# B&R Automation Studio project TD52 (part 44)

### Program Logical/Customized/c_red (IEC, version 4.11.0) - customisation task for exernal power reductions

#### c_redCyclic.st
```iecst
(*******************************************************************************
c_red 			customized power reductions

This code is confidential and proprietary to the INNIO Company.
It may not be used in any form, or reproduced in any manner,
without written permission of the INNIO Company.
Copyright, INNIO Company, 2021

Customized modifications: -
------------------------

History:
-------
V3.90.0	03.07.2012 Zengerer		new, (function moved from task gasum )
V4.02.0 ??.??.2015  ??			cleanup, separated INI file
V4.03.0	10.11.2015 Zengerer		cleanup
V4.04.0	08.03.2017 Zengerer		replace IN_CU.tCustAnaIn[1].Ai by a neutral IN_CU.tCustAnaIn[0].Ai default, to avoid conflicts when task is not used
V4.11.0	16.08.2021 Weitzer 		Delete W_XXmA constant variables

Instructions for use:
--------------------
connect var for customized spare power redutions

! ALL REDUCTIONS HAVE TO BE NORMED FROM 0 to 1 EQUALS 0 to P nominal

Outstandings:
------------
adopt this task according customer needs
replace [0] with actual used channel numbers IN_CU.tCustAnaIn[0].Ai;

*******************************************************************************)

PROGRAM _CYCLIC

	(*-----------------------------------------------------------------------------------------*)
	(*                                        TASK INPUTS                                      *)
	(*-----------------------------------------------------------------------------------------*)
 	OUT_CU.bP_Red_Sp_Lim1Act :=	FALSE;						(* CONNNECT REDUCTION ACTIVATION BIT HERE *)
	xSigScalR_Lim1Act.X := 		IN_CU.tCustAnaIn[0].Ai;		(* CONNNECT REDUCTION VALUE for customer spare power reduction, e.g. IN_CU.tCustAnaIn[1].Ai;	 *)
															(*hint: connect xSigScalR_Lim1Act.X1 and x2 also to available spare parameter*)

	OUT_CU.bP_Red_Sp_Lim2Act  	:= FALSE;					(* CONNNECT REDUCTION ACTIVATION BIT HERE *)
	xSigScalR_Lim2Act.X := 		IN_CU.tCustAnaIn[0].Ai;		(* CONNNECT REDUCTION VALUE for customer spare power reduction, e.g. IN_CU.tCustAnaIn[2].Ai; *)
															(*hint: connect xSigScalR_Lim2Act.X1 and x2 also to available spare parameter*)

	OUT_CU.bP_Red_Sp_Lim3Act  	:= FALSE;					(* CONNNECT REDUCTION ACTIVATION BIT HERE *)
	xSigScalR_Lim3Act.X := 		IN_CU.tCustAnaIn[0].Ai;		(* CONNNECT REDUCTION VALUE for customer spare power reduction, e.g. IN_CU.tCustAnaIn[3].Ai; *)
															(*hint: connect xSigScalR_Lim3Act.X1 and x2 also to available spare parameter*)

	(*-----------------------------------------------------------------------------------------*)
	(* Customer spare power reductions
	(*-----------------------------------------------------------------------------------------*)
	(* Reserve reduction #1 *)
	OUT_CU.bP_Red_Sp_Lim1Act; //:= FALSE;
	xSigScalR_Lim1Act.X; //		:= IN_CU.tCustAnaIn[x].Ai;
	xSigScalR_Lim1Act.X1 		:= Para.rCust_SparePara[0];		(* CONNNECT REDUCTION START VALUE, e.g. Para.rCust_SparePara[1]; *)
	xSigScalR_Lim1Act.Y1		:= 1.00;
	xSigScalR_Lim1Act.X2		:= Para.rCust_SparePara[0];		(* CONNNECT REDUCTION END VALUE, e.g. Para.rCust_SparePara[2];	 *)
	xSigScalR_Lim1Act.Y2		:= 0.50;
	xSigScalR_Lim1Act();
	IF OUT_CU.bP_Red_Sp_Lim1Act THEN
		OUT_CU.rP_Red_Sp_Lim1_Norm	:= LIMIT(0,xSigScalR_Lim1Act.Y_SCAL,1.0);
	ELSE
		OUT_CU.rP_Red_Sp_Lim1_Norm	:= 1.0;
	END_IF;

	(* Reserve reduction #2 *)
	OUT_CU.bP_Red_Sp_Lim2Act; //:= FALSE;
	xSigScalR_Lim2Act.X; //		:= IN_CU.tCustAnaIn[x].Ai;
	xSigScalR_Lim2Act.X1 		:= Para.rCust_SparePara[0];		(* CONNNECT REDUCTION START VALUE, e.g. Para.rCust_SparePara[1]; *)
	xSigScalR_Lim2Act.Y1		:= 1.00;
	xSigScalR_Lim2Act.X2		:= Para.rCust_SparePara[0];		(* CONNNECT REDUCTION END VALUE, e.g. Para.rCust_SparePara[2];	 *)
	xSigScalR_Lim2Act.Y2		:= 0.50;
	xSigScalR_Lim2Act();
	IF OUT_CU.bP_Red_Sp_Lim2Act THEN
		OUT_CU.rP_Red_Sp_Lim2_Norm	:= LIMIT(0,xSigScalR_Lim2Act.Y_SCAL,1.0);
	ELSE
		OUT_CU.rP_Red_Sp_Lim2_Norm	:= 1.0;
	END_IF;

	(* Reserve reduction #3 *)
	OUT_CU.bP_Red_Sp_Lim3Act; //:= FALSE;
	xSigScalR_Lim3Act.X	; //	:= IN_CU.tCustAnaIn[x].Ai;
	xSigScalR_Lim3Act.X1 		:= Para.rCust_SparePara[0];		(* CONNNECT REDUCTION START VALUE, e.g. Para.rCust_SparePara[1]; *)
	xSigScalR_Lim3Act.Y1		:= 1.00;
	xSigScalR_Lim3Act.X2		:= Para.rCust_SparePara[0];		(* CONNNECT REDUCTION END VALUE, e.g. Para.rCust_SparePara[2];	 *)
	xSigScalR_Lim3Act.Y2		:= 0.50;
	xSigScalR_Lim3Act();
	IF OUT_CU.bP_Red_Sp_Lim3Act THEN
		OUT_CU.rP_Red_Sp_Lim3_Norm	:= LIMIT(0,xSigScalR_Lim3Act.Y_SCAL,1.0);
	ELSE
		OUT_CU.rP_Red_Sp_Lim3_Norm	:= 1.0;
	END_IF;

	(*----------------------------------------------------------------------------------*)
	(* external utility(evu) request power reduction = iIdx_Pred_Type	:= neu25(31) *)
	(*----------------------------------------------------------------------------------*)
	(* Functionality MOVED TO MM GRID Code! *)

	(*----------------------------------------------------------------------------------*)
	(* limits for feedback signals to utility *)
	(*----------------------------------------------------------------------------------*)
	ton_RM_EVU[0](IN:= NOT IN_CU.tDI_Dem_P_Red_EVU_Stage1.Di AND NOT IN_CU.tDI_Dem_P_Red_EVU_Stage2.Di AND NOT IN_CU.tDI_Dem_P_Red_EVU_Stage3.Di AND IN_CU.bMCB_On , PT:= T#10s);	(* MCB_ON? -> to clarify...*)
	OUT_CU.tDO_P_Red_EVU_Stage0.Do := ton_RM_EVU[0].Q;		(* no power limit.and no lockout module *)

	lim_lo[1]( In:= IN_CU.rP_Act[1], Gw:= (Para.rP_Red_EVU_Stage1 + 0.01), Hy:= 0.01 );	(*OLD: lim_lo[1](In:= DINT_TO_INT((INT_TO_DINT(P_IST) * 1000)/ PN_GASART), Gw:= (ssPowRed_Utility_1 +10), Hy:= 10);*)
	ton_RM_EVU[1]( IN:= lim_lo[1].Q AND IN_CU.tDI_Dem_P_Red_EVU_Stage1.Di, PT:= T#30s );	(**)
	OUT_CU.tDO_P_Red_EVU_Stage1.Do := ton_RM_EVU[1].Q;		(* power limit.stage 1 (small reduction) *)

	lim_lo[2]( In:= IN_CU.rP_Act[1], Gw:= (Para.rP_Red_EVU_Stage2 + 0.01), Hy:= 0.01 );  (*OLD: lim_lo[2](In:= DINT_TO_INT((INT_TO_DINT(P_IST) * 1000)/ PN_GASART), Gw:= (ssPowRed_Utility_2 +10), Hy:= 10);*)
	ton_RM_EVU[2]( IN:= lim_lo[2].Q AND IN_CU.tDI_Dem_P_Red_EVU_Stage2.Di, PT:= T#30s );	(**)
	OUT_CU.tDO_P_Red_EVU_Stage2.Do := ton_RM_EVU[2].Q;		(* power limit.stage 2 (more reduction) *)

	lim_lo[3]( In:= IN_CU.rP_Act[1], Gw:= (Para.rP_Red_EVU_Stage3 + 0.01), Hy:= 0.01 );  (*OLD: lim_lo[3](In:= DINT_TO_INT((INT_TO_DINT(P_IST) * 1000)/ PN_GASART), Gw:= (ssPowRed_Utility_3 +10), Hy:= 10);*)
	ton_RM_EVU[3]( IN:= lim_lo[3].Q AND IN_CU.tDI_Dem_P_Red_EVU_Stage3.Di, PT:= T#30s );	(**)
	OUT_CU.tDO_P_Red_EVU_Stage3.Do := ton_RM_EVU[3].Q;		(* power limit.stage 3 (more reduction) *)

	lim_lo[4]( In:= IN_CU.rP_Act[1], Gw:= (Para.rP_Red_EVU_Stage4 + 0.01), Hy:= 0.01 );  (*OLD: lim_lo[4](In:= DINT_TO_INT((INT_TO_DINT(P_IST) * 1000)/ PN_GASART), Gw:= (ssPowRed_Utility_4 +10), Hy:= 10);*)
	ton_RM_EVU[4]( IN:= lim_lo[4].Q AND IN_CU.tDI_Dem_P_Red_EVU_Stage4.Di, PT:= T#30s );	(**)
	OUT_CU.tDO_P_Red_EVU_Stage4.Do := ton_RM_EVU[4].Q;		(* power limit.stage 4 (more reduction) *)

	lim_lo[5]( In:= IN_CU.rP_Act[1], Gw:= (Para.rP_Red_EVU_Stage5 + 0.01), Hy:= 0.01 );  (*OLD: lim_lo[?6?](In:= DINT_TO_INT((INT_TO_DINT(P_IST) * 1000)/ PN_GASART), Gw:= (ssPowRed_Utility_5 +10), Hy:= 10);*)
	ton_RM_EVU[5]( IN:= lim_lo[5].Q AND IN_CU.tDI_Dem_P_Red_EVU_Stage5.Di, PT:= T#30s );	(**)
	OUT_CU.tDO_P_Red_EVU_Stage5.Do := ton_RM_EVU[5].Q;		(*  (=most reduction)*)

	(*------------------------------------------------------------------------------------------*)
	(* generator: power factor controller dependent power reductions ??							*)
	(*------------------------------------------------------------------------------------------*)
	(* FUNCTION MOVED TO MODUL GENERATOR! *)

	(*-----------------------------------------------------------------------------------------*)
	(* power reduction for Extern – Analog (analog_dp):
	(*-----------------------------------------------------------------------------------------*)

	IF IN_CU.rP_Nom > 0 THEN
		rP_Red_AI_Norm := IN_CU.tP_Red_AI_Norm.Ai / IN_CU.rP_Nom;		(* parameter are entered in KW, so convert setpoint to Norm here    *)
	ELSE
		rP_Red_AI_Norm := 1.0;
	END_IF
			(* scaling (DISABELED HERE! NO additional scaling, allready done in the HAL (with customized parameter) *)
			Para.rI_P_Red_AI_NormScalMin;	Para.rI_P_Red_AI_NormScalMax;
			Para.rP_Red_AI_NormScalMin;		Para.rP_Red_AI_NormScalMax;

	(* power reduction on RSS Remote: (AFW_F)*)
	IF (IN_CU.iIdx_RSS = 2) AND IN_CU.tP_Red_AI_Norm.GoodQual THEN		(* locale representation of old AWS_F from IN_CU.iIdx_RSS = 2  *)
		OUT_CU.rP_Red_AI_Norm := LIMIT(0.5, rP_Red_AI_Norm, 1.0);		(*= analog power limit value *)
		OUT_CU.bP_Red_AI_Enable := TRUE ;
	ELSE
		OUT_CU.rP_Red_AI_Norm := 1.0;
		OUT_CU.bP_Red_AI_Enable := FALSE ;
	END_IF

	(*-----------------------------------------------------------------------------------------*)
	(*                                        TASK OUTPUTS                                     *)
	(*-----------------------------------------------------------------------------------------*)
	(* Prototype usage of all outputs: *)
	OUT_CU.bP_Red_Sp_Lim1Act ; 		(* power setpoint limit 1 activ *) (*OldName: bPowerSetpointLimit1; Cycle: 5;*)
	OUT_CU.bP_Red_Sp_Lim2Act ; 		(* power setpoint limit 2 activ *) (*OldName: bPowerSetpointLimit2; Cycle: 5;*)
	OUT_CU.bP_Red_Sp_Lim3Act ; 		(* power setpoint limit 3 activ *) (*OldName: bPowerSetpointLimit3; Cycle: 5;*)
	OUT_CU.rP_Red_Sp_Lim1_Norm ; 	(* power setpoint limit 1  related to rP_Nom *) (*OldName: ssPowerSetpointLimit1; Cycle: 5;*)
	OUT_CU.rP_Red_Sp_Lim2_Norm ; 	(* power setpoint limit 2  related to rP_Nom] *) (*OldName: ssPowerSetpointLimit2; Cycle: 5;*)
	OUT_CU.rP_Red_Sp_Lim3_Norm ; 	(* power setpoint limit 3  related to rP_Nom *) (*OldName: ssPowerSetpointLimit3; Cycle: 5;*)
	OUT_CU.bP_Red_EVU_Enable ; 		(* *) (*OldName: RED_EVU_Aktiv; Cycle: 5;*)
	OUT_CU.rP_Red_EVU_Norm ; 		(* power redutcion by utility *) (*OldName: RED_EVU; Cycle: 5;*)
	OUT_CU.rP_Red_AI_Norm ; 		(* power reduction by analog input *) (*OldName: ssPowerRedAnalog; Cycle: 5;*)

END_PROGRAM
```

#### c_redInit.st
```iecst
(********************************************************************
 * COPYRIGHT -- INNIO Company
 ********************************************************************
 * Programm: c_red
 * Datei: c_redInit.st
 * Autor: ZengereS
 * Erstellt: 24.Juni 2015
 ********************************************************************)

PROGRAM _INIT

	OUT_CU.rP_Red_EVU_Norm := 	1.0;	(*	ssExtPwrSetP4 ? *)

	OUT_CU.rP_Red_AI_Norm := 	1.0; 	(* power reduction by analog input *) (*OldName: ssPowerRedAnalog *)

	(* This factory default definition is only a backuü fallback solution. *)
	(* Set parameter values for normal operation in parameter file! *)
	ParaFactoryDefault.rP_Red_EVU_Stage1 := 		0.1;	(* [1/ P nom] *)
	ParaFactoryDefault.rP_Red_EVU_Stage2 := 		0.2;	(* [1/ P nom] *)
	ParaFactoryDefault.rP_Red_EVU_Stage3 := 		0.3;	(* [1/ P nom] *)
	ParaFactoryDefault.rP_Red_EVU_Stage4 := 		0.4;	(* [1/ P nom] *)
	ParaFactoryDefault.rP_Red_EVU_Stage5 := 		0.5;	(* [1/ P nom] *)

END_PROGRAM
```

#### c_red.var - Lokale Variablen
```iecst
(********************************************************************
 * COPYRIGHT -- INNIO Company
 ********************************************************************
 * Programm: c_red
 * Datei: c_red.var
 * Autor: ZengereS
 * Erstellt: 20. Februar 2013
 ********************************************************************
 * Lokale Variablen des Programms c_red
 ********************************************************************)
VAR
	ton_RM_EVU : ARRAY[0..5] OF TON;
	lim_lo : ARRAY[0..5] OF GR_MAXR;
	rP_Red_AI_Norm : REAL;
	xSigScalR_Lim1Act : xSigScal_R;
	xSigScalR_Lim2Act : xSigScal_R;
	xSigScalR_Lim3Act : xSigScal_R;
END_VAR
```

### Program Logical/Customized/c_set (IEC, version 4.13.0) - customisation task for external power setpoints

#### c_setCyclic.st
```iecst
(*******************************************************************************
c_set 			customized power SETPOINTS

This code is confidential and proprietary to the INNIO Company.
It may not be used in any form, or reproduced in any manner,
without written permission of the INNIO Company.
Copyright, INNIO Company, 2023

Customized modifications: -
------------------------

History:
-------
								History cleanup, Version based on V4.02.1	04.03.2015: prepared interface FOR different PI timing (->Caks Michael)
V4.03.0	12.11.2015 Zengerer		P_Set_ExtAI_Norm  changed fallback logic; REACTIVETED DI POWER SETPOINT LOGIC AND PARAMETER HERE! (since code IN GRID CODE task statGR HAS GOT A DIFFERENT FUNCTIONALITY
		22.12.2015 Ze/Caks		Para.bCA_IgnP_CylOffset_Active
V4.04.1 05.09.2017 zengerer		Nachziehen der Netzbezugsregler Änderungen von Schwab Christoph / Caks Michael aus File Bugs&Solution_MnsCtrl.zip
V4.04.5 10.10.2017 Zengerer		Update with interfaces from BASISUPDATE 4.04.00.05 iIdx_Pred_Type State
V4.05.0 10.10.2017 zengerer		prepared interface for adopted gasmixing setpoint at testbench or for customized applications
V4.05.1 07.03.2018 zengerer		cleanup
		30.01.2019 Hohensinner	added new interfaces to OP and GC
		20.03.2019 Hohensinner	Added external controller interface
V4.07.1	03.04.2019 Hohensinner	Added Parameter Info for new interfaces and comments
V4.09.0 22.01.2020 zengerer		avoid P setpoint switching with 0mA Value:	(IN_CU.tP_Set_ExtAI_Norm.GoodQual OR Para.rI_P_Set_ExtAI_NormScalMin < 0.004)
V4.10.0	16.10.2020 Weitzer 		Release of custom GCB synchronization demand OUT_CU.bCust_Dem_Sy and MCB re-synchronization demand OUT_CU.bCust_Dem_RSy added
		19.01.2021 Weitzer		Custom synchronization blocking added (OUT_CU.bBloc_SY_Rel_Cust)
		27.01.2021 Zengerer		TOF_N_Set_ExtAI_Norm_GoodQual T#12s delay,
		28.01.2021 Zengerer		power setpoint range limitation min #53
		12.03.2021 Zengerer		#262- Conditions internal or bus speed setpoint active for speed offset:	AND	(IN_CU.iMsg[2136]>0 OR IN_CU.iMsg[2137]>0)
V4.10.1	xx.08.2021 Ze, GruberK.	Issue #530 ...need N_Offset and not external setpoint; limit value to parameter values
V4.11.0	16.08.2021 Keller		External Droop Power setpoint (AI, Bus), iSource_F_N_OffsSet
V4.11.0	16.08.2021 Weitzer 		Delete W_XXmA constant variables
		21.01.2022 MayerR	    AI scaling and signal source selection for OUT_CU.rUset_Isl moved to GC module(v_ctr) and Bus interfaces (OUT_CU.rUset_Isl_Bus and OUT_CU.rQset_Droop_Bus) added
V4.11.1 31.05.2022 lettenb.		default setting OUT_CU.bCust_Dem_RSy := TRUE -> FALSE(RSy only in case of customer demand), bugfix
V4.12.0 22.01.2023 Zuschnig		H2 content via bus added
V4.13.0	25.05.2023 Zengerer 	Speed Setpoint limitation #1106
		24.08.2023 Zengerer		IN_CU.bMsg[xxxx] introduced
		16.10.2023 Bachler  	add OUT_CU.bOtherGeneratorsInLSL for bumpless transition to LSL
		20.11.2023 Farre		interfaces to SY, OP, GC, GR needed for Microgrid applications (2023-168)
		29.11.2023 Goenczi		add new interfaces to SY and OP

Instructions for use:
--------------------
connect var's for customized power setpoints

! ALL SETPOINTS HAVE TO BE NORMED FROM 0 to 1 EQUALS 0 to P nominal

Outstandings:
------------
TODO: CHECK NEW CUSTOMISED PARA vvm/addPLCtag

  adopt this task according customer needs

! Be aware, that several setpoints are also influenced from GRID CODE MODULE, if this is engaged !

*******************************************************************************)

PROGRAM _CYCLIC

	(*----------------------------------------------------------------------------------*)
	(* external DI request power setpoints *) (*REACTIVETED SETPOINT LOGIC AND PARAMETER HERE! (since code IN GRID CODE task statGR HAS GOT A NEW FUNCTIONALITY *)
	(*----------------------------------------------------------------------------------*)
	(* power setpoint according external request digital inputs *)
	IF    IN_CU.tP_GenC_SetFix5EU.Di	THEN
		OUT_CU.rP_Set_ExtDI_Cust_Norm	:=	LIMIT(0.4, Para.rP_Set5_ExtDI_Norm, 1.0); 	(*OldName: AW_EXPSH_DI; Cycle: 5;*)
	ELSIF IN_CU.tP_GenC_SetFix4EU.Di	THEN
		OUT_CU.rP_Set_ExtDI_Cust_Norm	:=	LIMIT(0.4, Para.rP_Set4_ExtDI_Norm, 1.0);
	ELSIF IN_CU.tP_GenC_SetFix3EU.Di	THEN
		OUT_CU.rP_Set_ExtDI_Cust_Norm	:=	LIMIT(0.4, Para.rP_Set3_ExtDI_Norm, 1.0);
	ELSIF IN_CU.tP_GenC_SetFix2EU.Di	THEN
		OUT_CU.rP_Set_ExtDI_Cust_Norm	:=	LIMIT(0.4, Para.rP_Set2_ExtDI_Norm, 1.0);
	ELSIF IN_CU.tP_GenC_SetFix1EU.Di	THEN
		OUT_CU.rP_Set_ExtDI_Cust_Norm	:=	LIMIT(0.4, Para.rP_Set1_ExtDI_Norm, 1.0);
	ELSE
		OUT_CU.rP_Set_ExtDI_Cust_Norm	:=	1.0;										(* replacement for rP_Set_ExtDI_Norm *)
	END_IF;

	OUT_CU.bP_Set_ExtDI_Enable := 	IN_CU.tP_GenC_SetFix1EU.Di OR
									IN_CU.tP_GenC_SetFix2EU.Di OR
									IN_CU.tP_GenC_SetFix3EU.Di OR
									IN_CU.tP_GenC_SetFix4EU.Di OR
									IN_CU.tP_GenC_SetFix5EU.Di;		(* or connect customized?*)

	(* power setpoint *)
	(******************)
	IF Para.bCtr_Mns_Enable AND IN_CU.tDem_Ctr_Mns.Di THEN
		rP_Set_ExtAI_Norm := OUT_CU.rP_Set_Mns_Norm;				(*old compatibility version, only for EngineController without rP_Set_Ctr_Mns_Norm*)
		OUT_CU.rP_Set_Ctr_Mns_Norm := OUT_CU.rP_Set_Mns_Norm;	(*new Interface V4.5, (in use for Ctr_Mns from V4.5 on)*)
		OUT_CU.bP_Set_Ctr_Mns_Enable := TRUE;					(*new Interface V4.5, (in use for Ctr_Mns from V4.5 on)*)
	ELSIF	IN_CU.rP_Nom > 0 THEN
		rP_Set_ExtAI_Norm := IN_CU.tP_Set_ExtAI_Norm.Ai / IN_CU.rP_Nom;		(* parameter are entered in KW, so convert Setpoint to Norm    *)
		OUT_CU.rP_Set_Ctr_Mns_Norm := rP_Set_ExtAI_Norm;
		OUT_CU.bP_Set_Ctr_Mns_Enable := FALSE;
	ELSE
		rP_Set_ExtAI_Norm := 1.0;
		OUT_CU.rP_Set_Ctr_Mns_Norm := rP_Set_ExtAI_Norm;
		OUT_CU.bP_Set_Ctr_Mns_Enable := FALSE;
	END_IF
			(* scaling (DISABELED HERE! NO additional scaling here, allready done in the HAL (with this customized parameter) *)
				Para.rI_P_Set_ExtAI_NormScalMin;	Para.rI_P_Set_ExtAI_NormScalMax;
				Para.rP_Set_ExtAI_NormScalMin;		Para.rP_Set_ExtAI_NormScalMax;

	IF 	(IN_CU.iIdx_OMSS = 2) AND 										(* =operating switch AUTO *)
		(IN_CU.iIdx_RSS = 2) AND 										(* =remote service selected *)
		(IN_CU.tP_Set_ExtAI_Norm.GoodQual								(* =analog input signal is ok *)
		  OR Para.rI_P_Set_ExtAI_NormScalMin < 0.004)
	THEN 																(* BWS_A AND Remote AND signal check is ok AND <deleted> *)
		OUT_CU.rP_Set_ExtAI_Norm := LIMIT(0.4,rP_Set_ExtAI_Norm, 1.0);	(*= analog power setpoint range limitation (V4.10 changed min)*)
		OUT_CU.bP_Set_ExtAI_Enable := TRUE ; 	 						(*OldName: AW_EXPSH_AI; Cycle: 5;*)
	ELSE
		OUT_CU.rP_Set_ExtAI_Norm := 0.50;								(*V4.03: changed fallback logic to standard min. load point*)
		OUT_CU.bP_Set_ExtAI_Enable := FALSE; 							(*OldName: AW_EXPSH_AI; Cycle: 5;*)
	END_IF

	(* speed setpoint *)
	(******************)
	IF Para.rN_EngNom > 0 THEN
		rN_Set_ExtAI_Norm := IN_CU.tN_Set_ExtAI_Norm.Ai / Para.rN_EngNom;		(* parameter are entered in KW, so convert Setpoint to Norm    *)
	ELSE
		rN_Set_ExtAI_Norm := 1.0;
	END_IF
			(* scaling (DISABELED HERE! No additional scaling here, allready done in the HAL (with this customized parameter) *)
			Para.rI_N_Set_ExtAI_NormScalMin;	Para.rI_N_Set_ExtAI_NormScalMax;
			Para.rN_Set_ExtAI_NormScalMin; 		Para.rN_Set_ExtAI_NormScalMax;

	TOF_N_Set_ExtAI_Norm_GoodQual(IN := IN_CU.tN_Set_ExtAI_Norm.GoodQual, PT := T#12s);		(*V4.10 delay*)
	IF  (IN_CU.iIdx_OMSS = 2) AND
		(IN_CU.iIdx_RSS = 2) AND
		TOF_N_Set_ExtAI_Norm_GoodQual.Q AND NOT
		(OUT_CU.iSource_F_N_OffsSet = 2) 			// typicaly needed N_Offset, not the external setpoint of previous default													(*V4.10 delay*)
//		IN_CU.tN_Set_ExtAI_Norm.GoodQual
// 		AND (Para.rI_N_Set_ExtAI_NormScalMin >0.004)
	THEN
		OUT_CU.rN_Set_ExtAI_Norm := LIMIT(0.9, rN_Set_ExtAI_Norm, 1.05);	(*= analog speed offset limitation  Limits adopted acc. issue #1106, 2023*)
		OUT_CU.bN_Set_ExtAI_Enable := TRUE ; (* *) 					(*OldName: AW_EX?SH_AI; Cycle: 5;*)
	ELSE
		OUT_CU.rN_Set_ExtAI_Norm := 1.0;
//		OUT_CU.bN_Set_ExtAI_Enable := FALSE ; (* *) 				(*OldName: AW_EX?SH_AI; Cycle: 5;*)
		OUT_CU.bN_Set_ExtAI_Enable := xOpMode.Island AND (Para.rI_N_Set_ExtAI_NormScalMin >0.004) AND TOF_N_Set_ExtAI_Norm_GoodQual.Q AND (OUT_CU.iSource_F_N_OffsSet = 2);  // Gruber K. - we need N_Offset and not external setpoint

	END_IF
				IN_CU.iMsg[2136]	;	(*display response: B2136 internal speed setpoint *)
 				IN_CU.iMsg[2137]	;	(*display response: B2137 external speed setpoint(bus) *)
				IN_CU.iMsg[2138]	;	(*display response: B2138 external speed setpoint(analoge) *)

	(******************************************************)
	(* Leistungsgrenzwert 1 - Customized z.b. ?Anforderung Lastabwurf? *)
	(*FEHLT NOCH:	GW_PGW1	   := DINT_TO_INT((INT_TO_DINT(PN_GASART) * Z_GW_PGW1  + 500) / 1000); *)
	Para.rP_Custom1_Norm_LimHi;		(* rP_Lim_Custom1_Norm == Z_GW_PGW1 = Para-Leistung-Grenzwerte-GRENZWERT 1 *)
	Para.rP_Custom1_Norm_HyHi;		(*FEHLT NOCH: 	HY_PGW1 ? Vorschlag  *)

(*FEHLT NOCH:	LAST_ABW :=  ( M_GSEIN AND NOT NS_EIN AND GW_PGW1 ) OR BL_OUT; *)	(*aus task pb8 -> wohin damit?*)

	(******************************************************)
	(* forwarding the parameter for different ignition timing on individual cylinders at testbench or for customized applications *)
	FOR ucCylinderCount := 1 TO 24 DO    (* bSetIndivTim can be used for tests                      *)
		IF IN_CU_ThisPlant.bCA_IgnP_ActiveMDE AND NOT IN_CU_ThisPlant.bMsg7000 THEN
			OUT_CU.rCA_IgnP_CylOffset[ucCylinderCount] := IN_CU_ThisPlant.rCA_IgnP_CylOffset_MDE[ucCylinderCount] * BOOL_TO_REAL(IN_CU_ThisPlant.bCA_IgnP_CylOffset_Active_MDE);
		ELSE
			OUT_CU.rCA_IgnP_CylOffset[ucCylinderCount] := Para.rCA_IgnP_CylOffset[ucCylinderCount] * BOOL_TO_REAL(Para.bCA_IgnP_CylOffset_Active);
		END_IF
	END_FOR

	(******************************************************)
	(* prepared interface for different PI timing on individual cylinders at testbench or for customized applications *)
     	OUT_CU.rCA_PI_Dur_COffset[1] := 0; 		(* custom PI duration offset cyl.1  *) (* OldName: ssTestBenchOffset *)
     	OUT_CU.rCA_PI_Dur_COffset[24] := 0; 	(* custom PI duration offset cyl.24 *) (* OldName: ssTestBenchOffset *)

	(******************************************************)
	(* prepared interface for adopted gasmixing setpoint *)
		OUT_CU.bOptGT_RatioMix_Set 	:= FALSE;   //:= TRUE;
 		OUT_CU.rGT_RatioMix_Set;				(* Fuel blending setpoint -> 0 - 1 = 0 - 100% )

	(******************************************************)

	(*** Enable bit for external speed / voltage controller ***)
	OUT_CU.bExtCtrOk := NOT IN_CU.tExtCtrOk.GoodQual OR IN_CU.tExtCtrOk.Di;		(* DI for use with ComAp or another external speed / voltage controller *)

	(*** Reactive power setpoint for voltage droop mode ***)
	(* Conversion:		1.0					100%Snom		*)
	(* Value range:		-1.0 to 1.0		-100% to 100%Snom	*)
	(* Build in Ramp:	0.01/s				1%Unom/s   		*)
	(* Enable:			Parameter 14298 must be set to 1	*)
	(* Droop gradient:	Parameter 14299						*)
	OUT_CU.rQset_Droop_Bus;									(* External reactive power setpoint for frequency droop mode over Bus - for project specific usage *)

	(* Voltage setpoint in Isolated operation, 0= no setpoint, 1= Droop, 2= External *)
	OUT_CU.rUset_Isl_Bus;									(* External Voltage setpoint (Island operation) over Bus - for project specific usage *)

	(*** Speed offset setpoint in Isolated operation ***)
	(* Conversion:		1.0					1 rpm			*)
	(* Value range:		-50	to +50			-50 to +50 rpm	*)
	(* Enable:			Parameter 14300 must be set to 2	*)
	IF IN_CU.tN_Set_ExtAI_Norm.GoodQual AND OUT_CU.bExtCtrOk THEN
		(* Check if value --> -50 to +50, Parameter 11781 should be -50 rpm & 11780 should be +50 rpm  *)
		IF		Para.rN_Set_ExtAI_NormScalMax < 150.0
			AND	Para.rN_Set_ExtAI_NormScalMin > -150.0
			//AND	(IN_CU.iMsg[2136]>0 OR IN_CU.iMsg[2137]>0)	// Gruber K. - will not work with this line included		(*V4.10: Offset allowed only at internal(2136) or bus(2137) speed setpoint, to avoid duplicate speed reduction in case of alternative input use *)
			AND NOT(IN_CU.tN_Set_ExtAI_Norm.Ai < -rN_Set_ExtAI_Limit OR IN_CU.tN_Set_ExtAI_Norm.Ai > rN_Set_ExtAI_Limit)(*V4.11: plausibility check *)
			THEN
				OUT_CU.rN_Offs_Cust		:=	LIMIT(Para.rN_Set_ExtAI_NormScalMin, IN_CU.tN_Set_ExtAI_Norm.Ai, Para.rN_Set_ExtAI_NormScalMax); (*Gruber K. - limit vlaue to parameter values*)
			(* Check if value --> 1450 to 1550, Parameter 11781 should be 0 or 1450 rpm & 11780 should be 1550 rpm *)
		ELSIF Para.rN_Set_ExtAI_NormScalMax > Para.rN_EngNom * 0.9 AND Para.rN_Set_ExtAI_NormScalMin < Para.rN_EngNom
			AND NOT(IN_CU.tN_Set_ExtAI_Norm.Ai < Para.rN_EngNom-rN_Set_ExtAI_Limit OR IN_CU.tN_Set_ExtAI_Norm.Ai > Para.rN_EngNom+rN_Set_ExtAI_Limit)(*V4.11: plausibility check *)
			THEN
			OUT_CU.rN_Offs_Cust		:=	IN_CU.tN_Set_ExtAI_Norm.Ai - Para.rN_EngNom;
			(* or implement your own solution *)							(* modify here if customer needs special scaling *)
		ELSE															(* modify here if customer needs special scaling *)
			OUT_CU.rN_Offs_Cust		:=	0.0;							(* modify here if customer needs special scaling *)
		END_IF
	ELSIF FALSE (*bN_OffsExt_Bus*) THEN									(* modify here if customer needs signal over bus *)
		OUT_CU.rN_Offs_Cust		:=	0.0;	(*rN_OffsExt_Bus*)			(* modify here if customer needs signal over bus *)
	ELSE
		OUT_CU.rN_Offs_Cust		:=	0.0;
	END_IF

	(*** Power setpoint for speed/frequency droop mode ***)
	(* Conversion:		1.0					100%Pnom		*)
	(* Value range:		0.0	to 1.0			0% to 100%Pnom	*)
	(* Build in Ramp:	Parameter 12095 & 13373	in %Pnom/s	*)
	(* Enable:			Parameter 14300 must be set to 1	*)
	(* Droop gradient:	Parameter 12109						*)
	OUT_CU.bP_Droop_Set_Bus;									(* Enable Droop power setpoint by Bus (if both true: has priority over AI)*)
	OUT_CU.bP_Droop_Set_AI; 									(* Enable Droop power setpoint by Analog input *)

	(** Fallback for power setpoint **)
	(* fallback if bP_Droop_Set_Bus = TRUE AND bus communication not OK *)
	(* fallback if bP_Droop_Set_AI = TRUE AND tP_Droop_Set.GoodQual = FALSE *)
	(* selection fallback mode, 0: default Para, 1: freeze last value*)
	OUT_CU.iIdx_Droop_SetDefaultCase 	:= Para.iIdx_Droop_SetDefaultCase;
	OUT_CU.rP_Set_Default_Norm 			:= Para.rP_Set_Default_Norm;

	(* Bus *)
	OUT_CU.rP_Droop_Set_Bus_Norm;(* HERE: implementation Droop setpoint bus interface *)
	IF NOT(IN_CU.bMsg[1147] OR IN_CU.bMsg[1099]) AND NOT(OUT_CU.rP_Droop_Set_Bus_Norm < -0.1 OR OUT_CU.rP_Droop_Set_Bus_Norm > 1.5) THEN
		rP_Droop_Set_Bus_old_Norm 		:= OUT_CU.rP_Droop_Set_Bus_Norm; 		(* save last valid setpoint *)
	ELSIF OUT_CU.iIdx_Droop_SetDefaultCase = 0 THEN
		OUT_CU.rP_Droop_Set_Bus_Norm	:= OUT_CU.rP_Set_Default_Norm;			(* 0: fallback, default parameter *)
	ELSIF OUT_CU.iIdx_Droop_SetDefaultCase = 1 THEN
		OUT_CU.rP_Droop_Set_Bus_Norm	:= rP_Droop_Set_Bus_old_Norm;			(* 1: fallback, freeze last valid setpoint *)
	ELSE
		OUT_CU.rP_Droop_Set_Bus_Norm	:= OUT_CU.rP_Set_Default_Norm;
	END_IF;

	(* Analog input *)
	IF IN_CU.tP_Droop_Set.GoodQual AND NOT(IN_CU.tP_Droop_Set.Ai < -0.1 OR IN_CU.tP_Droop_Set.Ai > 1.5) THEN
		OUT_CU.rP_Droop_Set_AI_Norm 	:= IN_CU.tP_Droop_Set.Ai;
		rP_Droop_Set_AI_old_Norm		:= OUT_CU.rP_Droop_Set_AI_Norm;  		(* save last valid setpoint *)
	ELSIF OUT_CU.iIdx_Droop_SetDefaultCase = 0 THEN
		OUT_CU.rP_Droop_Set_AI_Norm		:= OUT_CU.rP_Set_Default_Norm;			(* 0: fallback, default parameter *)
	ELSIF OUT_CU.iIdx_Droop_SetDefaultCase = 1 THEN
		OUT_CU.rP_Droop_Set_AI_Norm		:= rP_Droop_Set_AI_old_Norm;			(* 1: fallback, freeze last valid setpoint *)
	ELSE
		OUT_CU.rP_Droop_Set_AI_Norm 	:= OUT_CU.rP_Set_Default_Norm;
	END_IF;

	(* Load Sharing Mode, 0= no setpoint, 1= Droop, 2= External, 3= LSL *)
	OUT_CU.iSource_F_N_OffsSet := Para.iSource_F_N_OffsSet;
	MM2VIS.iSource_F_N_OffsSet := OUT_CU.iSource_F_N_OffsSet;

	(* Other Generators In Load Sharing Line *)
	(* If TRUE: 		Other engines are participating in the load sharing line *)
	(* Info: 			If this input is not provided a non smooth transition between LSL and the other load sharing modes will happen *)
	OUT_CU.bOtherGeneratorsInLSL;

	(*** Custom Engine demand ***)
	(* If TRUE:			Engine is demanded in AUTO & REMOTE	*)
	(* Info:			Add an Operating message why the engine is being demanded *)
	OUT_CU.bCust_Dem;

	(*** Custom Engine blocked ***)
	(* If TRUE:			Engine is blocked					*)
	(* Info:			If you want to block engine only in Stop mode use: 'bYourBit AND NOT bEng_StaSpdExc' *)
	OUT_CU.bEng_Block_Customized;

	(*Custom Emergency Power Supply release/demand*)

	(*** Release Island bit via Bus coupling ***)
	(* If FALSE:		Release island is blocked						*)
	(* Info:			Default value must be TRUE *)
	OUT_CU.bRel_I_Bus := TRUE;

	(*** Custom Release Island bit ***)
	(* If FALSE:		Release island is blocked						*)
	(* Info:			Default value must be TRUE *)
	OUT_CU.bCust_Rel_I := TRUE;

	(*** Custom Release Island operation busbar condition (if FALSE, mains cut-off with gcb) ***)
	(* If TRUE:			VKE10 condition TRUE					*)
	(* Info:			DO NOT CONFUSE WITH bRel_I Release island external bit!!! --- Default value must be FALSE *)
	OUT_CU.bCust_RelI_BB := FALSE;

	(*** Custom Emergency Power supply demand SY modul ***)
	(* If TRUE:			Additional demand condition to change to EPS mode in SY/sy_out task				*)
	(* Info:			Default value must be TRUE *)
	OUT_CU.bCust_Dem_EPS_Sy := TRUE;

	(*** External Emergency Power supply demand from Bus ***)
	(* If TRUE:			Emergency Power supply ON				*)
	(* Info:			Default value must be FALSE *)
	OUT_CU.bEng_Dem_EPS_Bus := FALSE;

	(*** Smooth engine discharge in multi engines island mode ***)
	(* If TRUE:			Engine is not demanded for island, request auto blocked, but release island is still active -
						engine runs until P_Lo reached and GCB opens - other genset has to be demanded and on (GCB_OGP) to take load + on site load shedding device					*)
	(* Info:			For single engine it is FALSE as EngDemIsland label does not exist, *)
	OUT_CU.bSmoothDischarge_CU := NOT bOMSS_Man	AND NOT IN_CU.tEngDemIsland.Di;

	(* CH4 signal from BUS system *)
	(* If TRUE:			CH4 signal is sent via bus if parameter [11364] is active 				*)
	OUT_CU.bCH4_Bus_Active;
	(* Info:			CH4 signal - 1.0 = 100%													*)
	OUT_CU.rCH4_Bus;

	(* H2 signal from BUS system *)
	(* If TRUE:			H2 signal is sent via bus if parameter [14901] is active 				*)
	OUT_CU.bH2_Bus_Active;
	(* Info:			H2 signal - 1.0 = 100%													*)
	OUT_CU.rH2_Bus;
	(* If FALSE:		Measurement signal failure H2 content if OUT_CU.bH2_Bus_Active active	*)
	OUT_CU.bH2_Bus_MSF;

	(* CV signal from BUS system *)
	(* If TRUE:			CV signal is sent via bus if parameter [11367] is active 				*)
	OUT_CU.bCV_Bus_Active;
	(* Info:			CV signal in [kWh/Nm3]													*)
	OUT_CU.rCV_Bus;

	(* Info:			Calibration signal from bus or IN_GT.tGT_CalibrateActive.Di can be used *)
	OUT_CU.bGT_CalibrateActive_Bus;

	(* Release gas plant signal from BUS system *)
	(* If TRUE:			Release gas plant signal is sent via bus 				 				*)
	OUT_CU.bRelGasPlant_Bus_Active;
	(* If FALSE:			Release from gas plant missing										*)
	OUT_CU.bRelGasPlant_Bus;

	(* External Synchroniszation by Customer *)

	(*** Custom GCB synchronization demand     ***)
	(* If TRUE:			GCB Sync is released	 *)
	(* Info:									 *)
	OUT_CU.bCust_Dem_Sy := TRUE;

	(*** Custom MCB re-synchronization demand  ***)
	(* If TRUE:			MCB Re-Sync is released  *)
	(* Info:			 						 *)
	OUT_CU.bCust_Dem_RSy := FALSE;

	(*** Custom synchronization blocking         ***)
	(* If TRUE:			synchronisation is blocked *)
	(* Info:			 						   *)
	OUT_CU.bBloc_SY_Rel_Cust := FALSE;

	(*** Microgrid Interfaces to SY, GC, GR, OP   ***)
	(* Bypass MCB status - dead busbar *)
	OUT_CU.bBypassMCB_deadBB 	:= FALSE;
	(* Bypass MCB status - soft energisation *)
	OUT_CU.bSoftEnergDem	 	:= FALSE;
	OUT_CU.bBypassMCB_SoftStart := FALSE;
	(* Bypass MCB status - load shedding *)
	OUT_CU.bBypassMCB_LoadShed	:= FALSE;
	(* Bypass MCB status - Cos Phi Ctrl *)
	OUT_CU.bBypassMCB_CosPhi	:= FALSE;
	(* Bypass MCB status - FSM *)
	OUT_CU.bBypassMCB_FSM		:= FALSE;
	(* Dead band definition for FSM/LFSM *)
	OUT_CU.bDroopDB_Active	    := FALSE;
	OUT_CU.rDB_FSM_LFSM			:= 0.5; //standard value
	(* request power mode *)
	OUT_CU.bReq_PowMod := IN_CU.tReq_PowMod.Di;
	(* extended power operation range *)
	OUT_CU.bExtendedOpRangeRel	:= FALSE;
	OUT_CU.rP_Set_Min_Norm_Ext	:= 0.5; (* !! rP_Set_Min_Norm internally limited to 10% !!*)

	(* Engine calibration TO EC - PVcheckNEW - ONLY USE AFTER AGREEMENT WITH SYSTEM OWNER EC!!! *)
	OUT_CU.iAggrekoEngineVersion 	:= 0;				(* Aggreko egine version: 1 = J420B, 2 = J420C, 3 = J420E *)
	OUT_CU.iAggrekoTCConfig		:= 0;				(* Aggreko CBV configuration: 1 = TA40, 2 = TA45, 3 = TA65 *)

END_PROGRAM
```

#### c_setInit.st
```iecst
(********************************************************************
 * COPYRIGHT -- INNIO Company
 ********************************************************************
 * Programm: c_set
 * Datei: c_setInit.st
 * Autor: ZengereS
 * Erstellt: 2. April 2013
 ********************************************************************
 * Implementierung des Programms c_set
 ********************************************************************)

PROGRAM _INIT

	 IN_CU.tP_Set_ExtAI_Norm.Ai :=	1.0;
//	 IN_CU.tN_Set_ExtAI_Norm.Ai :=	1.0;

	(*----------------------------------------------------------------------------------*)
	(* Prototype usage and predifinition of all outputs: *)
	OUT_CU.bP_Set_ExtDI_Enable := 	FALSE ; (* *)  	(*OldName: AW_EXPSH_DI; Cycle: 5;*)
	//OUT_CU.rP_Set_ExtDI_Norm :=		1.0;	(* *) 	(*OldName: Dig_P_SOLL; Cycle: 5;*)  (*REMOVE SETPOINTS HERE, AS SOON AS THEIR FUNCTIONALITY IS PROVIDED BY GRID CODE LOGIC*)

	OUT_CU.bP_Set_ExtAI_Enable := 	FALSE ; (* *) 	(*OldName: AW_EXPSH_AI; Cycle: 5;*)
	OUT_CU.rP_Set_ExtAI_Norm := 	1.0;	(* *) 	(*OldName: ssNominalPowerAnalog		; Cycle: 5;*)
	OUT_CU.bN_Set_ExtAI_Enable := 	FALSE ; (* *) 	(*OldName: AW_EXDSH; Cycle: 5;*)
	OUT_CU.rN_Set_ExtAI_Norm := 	1.0;	(* *) 	(*OldName: Dig_N_SOLL; Cycle: 5;*)

	(*OLD Varnames, Do not use anymore - soon o be deleted:*)
	sel_PowerSetpointLimit ; 	(*(Varname Old for compatibility)*)
	bPowerSetpointLimit ; 		(*(Varname Old for compatibility)*)
	ssPowerSetpointLimit ; 		(*(Varname Old for compatibility)*)

	IF Para.rN_EngNom = 0 THEN Para.rN_EngNom := 1500.1;	END_IF		(*Fallback for missing parameter AdditionalPLCTag*)

END_PROGRAM
```

#### c_set.var - Lokale Variablen
```iecst
(********************************************************************
 * COPYRIGHT -- INNIO Company
 ********************************************************************
 * Programm: c_red
 * Datei: c_red.var
 * Autor: ZengereS
 * Erstellt: 20. Februar 2013
 ********************************************************************
 * Lokale Variablen des Programms c_red
 ********************************************************************)
VAR
	rP_Set_ExtAI_Norm : REAL;
	rN_Set_ExtAI_Norm : REAL;
	ucCylinderCount : USINT;
	TOF_N_Set_ExtAI_Norm_GoodQual : TOF := (0);
	rP_Droop_Set_Bus_old_Norm : REAL := 0.0; (*Droop Fallback mode 1: freezed setpoint value BUS [-]*)
	rP_Droop_Set_AI_old_Norm : REAL := 0.0; (*Droop Fallback mode 1: freezed setpoint value [-] AI*)
	rN_Set_ExtAI_Limit : REAL := 50; (*External speed offset limit in rpm (+-)*)
END_VAR
```

### Program Logical/Customized/c_dig (IEC, version 4.07.0) - Digital I/O Task to handle prepared customizable digital signals

#### c_digCyclic.st
```iecst
(*******************************************************************************
CUSTOMIZED: c_dig.st - connection and processing of prepared digital I /O channels (cyclic)

This code is confidential and proprietary to the INNIO Company.
It may not be used in any form, or reproduced in any manner, without the express
written permission of the INNIO Company.
Copyright, INNIO Company, 2019

Customized modifications:
------------------------

History:
-------
V3.90	13.12.2012 Zengerer	NEW
...
V4.02.0 24.06.2015 Zengerer 	cleanup
V4.03.0	18.12.2015 Zengerer 	Bugfix Version for missing VIS parameter: Set all DigOut as active
		09.05.2016 lettenb.		Para.bCustDigOut_Active[x] entfernt, weil nicht in visu ausgeführt
		03.06.2016 lettenb.		IN_CU.tCustDigIn[41-60].Di removed (doppelt codiert)
V4.04.0	16.06.2016 Weitzer		add CustDigIn[81..200]
V4.07.0 19.12.2018 Zengerer		add IN_CU.tCustDigIn_TC2[] with TaskClass2 .vvm

Instructions for use:
--------------------
- connect (or replace) <bConnectYourBitHere> with plant specific variables
- mark used channels here, to avoid duplicate usage withhin one customer project

AVOID HARDCODED Para.xxx VALUES!
You MAYBE want to enter SOME factory default values in the INIT section, but ONLY TO THE Para_FactoryDefault.xxx STRUCTURE!
By this way the parameter values in Para.xxx would stay acessible according to XT4 parameter management process.

Outstandings:
------------

*********************************************************************************)

PROGRAM _CYCLIC

	(*********************************************************************************************************************************)

	(********************************************************)
	(*                                                      *)
	(*                 DIGITAL INPUT SECTION                *)
	(*                                                      *)
	(********************************************************)

//	(* Reservedigitaleingang x *)									(* (KONFIGURATIONSBEISPIEL)*)
//	(* reserve digital input x *)									(* (CONFIGURATION EXAMPLE) *)
//	(***************************)
//	bConnectYourBitHere		:= IN_CU.tCustDigIn[x].Di;		(*Anpassen entsprechend Kundenanforderung*)	 			(* change 'bConnectYourBitHere' customized *)
//							   IN_CU.tCustDigIn_TC2[x].Di; 	(*reminder: for fast counter inputs in TC#2 tasks use IN_CU.tCustDigIn_TC2[] directly!   *)
//	OUT_CU.bCustDigIn[x]	:= IN_CU.tCustDigIn[x].Di;		(*Vorbereitete OUT- Modulschnittst. (braucht .vvm)*)	(* modul OUT interface is prepared for possible usage of this input value in other modules	(edit other module´s .vvm, if necessary)*)
//	MM2VIS.bCustDigIn[x]	:= IN_CU.tCustDigIn[x].Di;		(*Dies Variabele iat für die VIS Verwendung vorber.*)	(* prepared for VIS	usage *)

	(* reserve digital input 1 *)
	bConnectYourBitHere		:= IN_CU.tCustDigIn[1].Di;
							   IN_CU.tCustDigIn_TC2[1].Di; 	(*reminder: for fast counter inputs in TC#2 tasks use IN_CU.tCustDigIn_TC2[] directly!  (V4.07) *)
	OUT_CU.bCustDigIn[1]	:= IN_CU.tCustDigIn[1].Di;		(*stated here only once as reminder, processing is done in loop*)
	MM2VIS.bCustDigIn[1]	:= IN_CU.tCustDigIn[1].Di;		(*stated here only once as reminder, processing is done in loop*)
	(* reserve digital input 2 *)
	bConnectYourBitHere		:= IN_CU.tCustDigIn[2].Di;
	(* reserve digital input 3 *)
	bConnectYourBitHere		:= IN_CU.tCustDigIn[3].Di;
	(* reserve digital input 4 *)
	bConnectYourBitHere		:= IN_CU.tCustDigIn[4].Di;

	(* reserve digital input 5 *)
	bConnectYourBitHere		:= IN_CU.tCustDigIn[5].Di;
	(* reserve digital input 6 *)
	bConnectYourBitHere		:= IN_CU.tCustDigIn[6].Di;
	(* reserve digital input 7 *)
	bConnectYourBitHere		:= IN_CU.tCustDigIn[7].Di;
	(* reserve digital input 8 *)
	bConnectYourBitHere		:= IN_CU.tCustDigIn[8].Di;

	(* reserve digital input 9 *)
	bConnectYourBitHere		:= IN_CU.tCustDigIn[9].Di;
	(* reserve digital input 10 *)
	bConnectYourBitHere		:= IN_CU.tCustDigIn[10].Di;
	(* reserve digital input 11 *)
	bConnectYourBitHere		:= IN_CU.tCustDigIn[11].Di;
	(* reserve digital input 12 *)
	bConnectYourBitHere		:= IN_CU.tCustDigIn[12].Di;

	(* reserve digital input 13 *)
	bConnectYourBitHere		:= IN_CU.tCustDigIn[13].Di;
	bConnectYourBitHere		:= IN_CU.tCustDigIn[14].Di;
	bConnectYourBitHere		:= IN_CU.tCustDigIn[15].Di;
	bConnectYourBitHere		:= IN_CU.tCustDigIn[16].Di;

	(* reserve digital input 17 *)
	bConnectYourBitHere		:= IN_CU.tCustDigIn[17].Di;
	bConnectYourBitHere		:= IN_CU.tCustDigIn[18].Di;
	bConnectYourBitHere		:= IN_CU.tCustDigIn[19].Di;
	bConnectYourBitHere		:= IN_CU.tCustDigIn[20].Di;

	(* reserve digital input 21 *)
	bConnectYourBitHere		:= IN_CU.tCustDigIn[21].Di;
	bConnectYourBitHere		:= IN_CU.tCustDigIn[22].Di;
	bConnectYourBitHere		:= IN_CU.tCustDigIn[23].Di;
	bConnectYourBitHere		:= IN_CU.tCustDigIn[24].Di;

	(* reserve digital input 25 *)
	bConnectYourBitHere		:= IN_CU.tCustDigIn[25].Di;
	bConnectYourBitHere		:= IN_CU.tCustDigIn[26].Di;
	bConnectYourBitHere		:= IN_CU.tCustDigIn[27].Di;
	bConnectYourBitHere		:= IN_CU.tCustDigIn[28].Di;

	(* reserve digital input 29 *)
	bConnectYourBitHere		:= IN_CU.tCustDigIn[29].Di;
	bConnectYourBitHere		:= IN_CU.tCustDigIn[30].Di;
	bConnectYourBitHere		:= IN_CU.tCustDigIn[31].Di;
	bConnectYourBitHere		:= IN_CU.tCustDigIn[32].Di;

	(* reserve digital input 33 *)
	bConnectYourBitHere		:= IN_CU.tCustDigIn[33].Di;
	bConnectYourBitHere		:= IN_CU.tCustDigIn[34].Di;
	bConnectYourBitHere		:= IN_CU.tCustDigIn[35].Di;
	bConnectYourBitHere		:= IN_CU.tCustDigIn[36].Di;

	(* reserve digital input 37 *)
	bConnectYourBitHere		:= IN_CU.tCustDigIn[37].Di;
	bConnectYourBitHere		:= IN_CU.tCustDigIn[38].Di;
	bConnectYourBitHere		:= IN_CU.tCustDigIn[39].Di;
	bConnectYourBitHere		:= IN_CU.tCustDigIn[40].Di;

	(* reserve digital input 41 *)
	bConnectYourBitHere		:= IN_CU.tCustDigIn[41].Di;
	bConnectYourBitHere		:= IN_CU.tCustDigIn[42].Di;
	bConnectYourBitHere		:= IN_CU.tCustDigIn[43].Di;
	bConnectYourBitHere		:= IN_CU.tCustDigIn[44].Di;

	(* reserve digital input 45 *)
	bConnectYourBitHere		:= IN_CU.tCustDigIn[45].Di;
	bConnectYourBitHere		:= IN_CU.tCustDigIn[46].Di;
	bConnectYourBitHere		:= IN_CU.tCustDigIn[47].Di;
	bConnectYourBitHere		:= IN_CU.tCustDigIn[48].Di;

	(* reserve digital input 49 *)
	bConnectYourBitHere		:= IN_CU.tCustDigIn[49].Di;
	bConnectYourBitHere		:= IN_CU.tCustDigIn[50].Di;
	bConnectYourBitHere		:= IN_CU.tCustDigIn[51].Di;
	bConnectYourBitHere		:= IN_CU.tCustDigIn[52].Di;

	(* reserve digital input 53 *)
	bConnectYourBitHere		:= IN_CU.tCustDigIn[53].Di;
	bConnectYourBitHere		:= IN_CU.tCustDigIn[54].Di;
	bConnectYourBitHere		:= IN_CU.tCustDigIn[55].Di;
	bConnectYourBitHere		:= IN_CU.tCustDigIn[56].Di;

	(* reserve digital input 57 *)
	bConnectYourBitHere		:= IN_CU.tCustDigIn[57].Di;
	bConnectYourBitHere		:= IN_CU.tCustDigIn[58].Di;
	bConnectYourBitHere		:= IN_CU.tCustDigIn[59].Di;
	bConnectYourBitHere		:= IN_CU.tCustDigIn[60].Di;

	(* reserve digital input 61 *)
	bConnectYourBitHere		:= IN_CU.tCustDigIn[61].Di;
	bConnectYourBitHere		:= IN_CU.tCustDigIn[62].Di;
	bConnectYourBitHere		:= IN_CU.tCustDigIn[63].Di;
	bConnectYourBitHere		:= IN_CU.tCustDigIn[64].Di;

	(* reserve digital input 65 *)
	bConnectYourBitHere		:= IN_CU.tCustDigIn[65].Di;
	bConnectYourBitHere		:= IN_CU.tCustDigIn[66].Di;
	bConnectYourBitHere		:= IN_CU.tCustDigIn[67].Di;
	bConnectYourBitHere		:= IN_CU.tCustDigIn[68].Di;

	(* reserve digital input 69 *)
	bConnectYourBitHere		:= IN_CU.tCustDigIn[69].Di;
	bConnectYourBitHere		:= IN_CU.tCustDigIn[70].Di;
	bConnectYourBitHere		:= IN_CU.tCustDigIn[71].Di;
	bConnectYourBitHere		:= IN_CU.tCustDigIn[72].Di;

	(* reserve digital input 73 *)
	bConnectYourBitHere		:= IN_CU.tCustDigIn[73].Di;
	bConnectYourBitHere		:= IN_CU.tCustDigIn[74].Di;
	bConnectYourBitHere		:= IN_CU.tCustDigIn[75].Di;
	bConnectYourBitHere		:= IN_CU.tCustDigIn[76].Di;

	(* reserve digital input 77 *)
	bConnectYourBitHere		:= IN_CU.tCustDigIn[77].Di;
	bConnectYourBitHere		:= IN_CU.tCustDigIn[78].Di;
	bConnectYourBitHere		:= IN_CU.tCustDigIn[79].Di;
	bConnectYourBitHere		:= IN_CU.tCustDigIn[80].Di;

	(* reserve digital input 81 *)
	bConnectYourBitHere		:= IN_CU.tCustDigIn[81].Di;
	bConnectYourBitHere		:= IN_CU.tCustDigIn[82].Di;
	bConnectYourBitHere		:= IN_CU.tCustDigIn[83].Di;
	bConnectYourBitHere		:= IN_CU.tCustDigIn[84].Di;

	(* reserve digital input 85 *)
	bConnectYourBitHere		:= IN_CU.tCustDigIn[85].Di;
	bConnectYourBitHere		:= IN_CU.tCustDigIn[86].Di;
	bConnectYourBitHere		:= IN_CU.tCustDigIn[87].Di;
	bConnectYourBitHere		:= IN_CU.tCustDigIn[88].Di;

	(* reserve digital input 89 *)
	bConnectYourBitHere		:= IN_CU.tCustDigIn[89].Di;
	bConnectYourBitHere		:= IN_CU.tCustDigIn[90].Di;
	bConnectYourBitHere		:= IN_CU.tCustDigIn[91].Di;
	bConnectYourBitHere		:= IN_CU.tCustDigIn[92].Di;

	(* reserve digital input 93 *)
	bConnectYourBitHere		:= IN_CU.tCustDigIn[93].Di;
	bConnectYourBitHere		:= IN_CU.tCustDigIn[94].Di;
	bConnectYourBitHere		:= IN_CU.tCustDigIn[95].Di;
	bConnectYourBitHere		:= IN_CU.tCustDigIn[96].Di;

	(* reserve digital input 97 *)
	bConnectYourBitHere		:= IN_CU.tCustDigIn[97].Di;
	bConnectYourBitHere		:= IN_CU.tCustDigIn[98].Di;
	bConnectYourBitHere		:= IN_CU.tCustDigIn[99].Di;
	bConnectYourBitHere		:= IN_CU.tCustDigIn[100].Di;

	(* reserve digital input 101 *)
	bConnectYourBitHere		:= IN_CU.tCustDigIn[101].Di;
	bConnectYourBitHere		:= IN_CU.tCustDigIn[102].Di;
	bConnectYourBitHere		:= IN_CU.tCustDigIn[103].Di;
	bConnectYourBitHere		:= IN_CU.tCustDigIn[104].Di;

	(* reserve digital input 105 *)
	bConnectYourBitHere		:= IN_CU.tCustDigIn[105].Di;
	bConnectYourBitHere		:= IN_CU.tCustDigIn[106].Di;
	bConnectYourBitHere		:= IN_CU.tCustDigIn[107].Di;
	bConnectYourBitHere		:= IN_CU.tCustDigIn[108].Di;

	(* reserve digital input 109 *)
	bConnectYourBitHere		:= IN_CU.tCustDigIn[109].Di;
	bConnectYourBitHere		:= IN_CU.tCustDigIn[110].Di;
	bConnectYourBitHere		:= IN_CU.tCustDigIn[111].Di;
	bConnectYourBitHere		:= IN_CU.tCustDigIn[112].Di;

	(* reserve digital input 113 *)
	bConnectYourBitHere		:= IN_CU.tCustDigIn[113].Di;
	bConnectYourBitHere		:= IN_CU.tCustDigIn[114].Di;
	bConnectYourBitHere		:= IN_CU.tCustDigIn[115].Di;
	bConnectYourBitHere		:= IN_CU.tCustDigIn[116].Di;

	(* reserve digital input 117 *)
	bConnectYourBitHere		:= IN_CU.tCustDigIn[117].Di;
	bConnectYourBitHere		:= IN_CU.tCustDigIn[118].Di;
	bConnectYourBitHere		:= IN_CU.tCustDigIn[119].Di;
	bConnectYourBitHere		:= IN_CU.tCustDigIn[120].Di;

	(* reserve digital input 121 *)
	bConnectYourBitHere		:= IN_CU.tCustDigIn[121].Di;
	bConnectYourBitHere		:= IN_CU.tCustDigIn[122].Di;
	bConnectYourBitHere		:= IN_CU.tCustDigIn[123].Di;
	bConnectYourBitHere		:= IN_CU.tCustDigIn[124].Di;

	(* reserve digital input 125 *)
	bConnectYourBitHere		:= IN_CU.tCustDigIn[125].Di;
	bConnectYourBitHere		:= IN_CU.tCustDigIn[126].Di;
	bConnectYourBitHere		:= IN_CU.tCustDigIn[127].Di;
	bConnectYourBitHere		:= IN_CU.tCustDigIn[128].Di;

	(* reserve digital input 129 *)
	bConnectYourBitHere		:= IN_CU.tCustDigIn[129].Di;
	bConnectYourBitHere		:= IN_CU.tCustDigIn[130].Di;
	bConnectYourBitHere		:= IN_CU.tCustDigIn[131].Di;
	bConnectYourBitHere		:= IN_CU.tCustDigIn[132].Di;

	(* reserve digital input 133 *)
	bConnectYourBitHere		:= IN_CU.tCustDigIn[133].Di;
	bConnectYourBitHere		:= IN_CU.tCustDigIn[134].Di;
	bConnectYourBitHere		:= IN_CU.tCustDigIn[135].Di;
	bConnectYourBitHere		:= IN_CU.tCustDigIn[136].Di;

	(* reserve digital input 137 *)
	bConnectYourBitHere		:= IN_CU.tCustDigIn[137].Di;
	bConnectYourBitHere		:= IN_CU.tCustDigIn[138].Di;
	bConnectYourBitHere		:= IN_CU.tCustDigIn[139].Di;
	bConnectYourBitHere		:= IN_CU.tCustDigIn[140].Di;

	(* reserve digital input 141 *)
	bConnectYourBitHere		:= IN_CU.tCustDigIn[141].Di;
	bConnectYourBitHere		:= IN_CU.tCustDigIn[142].Di;
	bConnectYourBitHere		:= IN_CU.tCustDigIn[143].Di;
	bConnectYourBitHere		:= IN_CU.tCustDigIn[144].Di;

	(* reserve digital input 145 *)
	bConnectYourBitHere		:= IN_CU.tCustDigIn[145].Di;
	bConnectYourBitHere		:= IN_CU.tCustDigIn[146].Di;
	bConnectYourBitHere		:= IN_CU.tCustDigIn[147].Di;
	bConnectYourBitHere		:= IN_CU.tCustDigIn[148].Di;

	(* reserve digital input 149 *)
	bConnectYourBitHere		:= IN_CU.tCustDigIn[149].Di;
	bConnectYourBitHere		:= IN_CU.tCustDigIn[150].Di;
	bConnectYourBitHere		:= IN_CU.tCustDigIn[151].Di;
	bConnectYourBitHere		:= IN_CU.tCustDigIn[152].Di;

	(* reserve digital input 153 *)
	bConnectYourBitHere		:= IN_CU.tCustDigIn[153].Di;
	bConnectYourBitHere		:= IN_CU.tCustDigIn[154].Di;
	bConnectYourBitHere		:= IN_CU.tCustDigIn[155].Di;
	bConnectYourBitHere		:= IN_CU.tCustDigIn[156].Di;

	(* reserve digital input 157 *)
	bConnectYourBitHere		:= IN_CU.tCustDigIn[157].Di;
	bConnectYourBitHere		:= IN_CU.tCustDigIn[158].Di;
	bConnectYourBitHere		:= IN_CU.tCustDigIn[159].Di;
	bConnectYourBitHere		:= IN_CU.tCustDigIn[160].Di;

	(* reserve digital input 161 *)
	bConnectYourBitHere		:= IN_CU.tCustDigIn[161].Di;
	bConnectYourBitHere		:= IN_CU.tCustDigIn[162].Di;
	bConnectYourBitHere		:= IN_CU.tCustDigIn[163].Di;
	bConnectYourBitHere		:= IN_CU.tCustDigIn[164].Di;

	(* reserve digital input 165 *)
	bConnectYourBitHere		:= IN_CU.tCustDigIn[165].Di;
	bConnectYourBitHere		:= IN_CU.tCustDigIn[166].Di;
	bConnectYourBitHere		:= IN_CU.tCustDigIn[167].Di;
	bConnectYourBitHere		:= IN_CU.tCustDigIn[168].Di;

	(* reserve digital input 169 *)
	bConnectYourBitHere		:= IN_CU.tCustDigIn[169].Di;
	bConnectYourBitHere		:= IN_CU.tCustDigIn[170].Di;
	bConnectYourBitHere		:= IN_CU.tCustDigIn[171].Di;
	bConnectYourBitHere		:= IN_CU.tCustDigIn[172].Di;

	(* reserve digital input 173 *)
	bConnectYourBitHere		:= IN_CU.tCustDigIn[173].Di;
	bConnectYourBitHere		:= IN_CU.tCustDigIn[174].Di;
	bConnectYourBitHere		:= IN_CU.tCustDigIn[175].Di;
	bConnectYourBitHere		:= IN_CU.tCustDigIn[176].Di;

	(* reserve digital input 177 *)
	bConnectYourBitHere		:= IN_CU.tCustDigIn[177].Di;
	bConnectYourBitHere		:= IN_CU.tCustDigIn[178].Di;
	bConnectYourBitHere		:= IN_CU.tCustDigIn[179].Di;
	bConnectYourBitHere		:= IN_CU.tCustDigIn[180].Di;

	(* reserve digital input 181 *)
	bConnectYourBitHere		:= IN_CU.tCustDigIn[181].Di;
	bConnectYourBitHere		:= IN_CU.tCustDigIn[182].Di;
	bConnectYourBitHere		:= IN_CU.tCustDigIn[183].Di;
	bConnectYourBitHere		:= IN_CU.tCustDigIn[184].Di;

	(* reserve digital input 185 *)
	bConnectYourBitHere		:= IN_CU.tCustDigIn[185].Di;
	bConnectYourBitHere		:= IN_CU.tCustDigIn[186].Di;
	bConnectYourBitHere		:= IN_CU.tCustDigIn[187].Di;
	bConnectYourBitHere		:= IN_CU.tCustDigIn[188].Di;

	(* reserve digital input 189 *)
	bConnectYourBitHere		:= IN_CU.tCustDigIn[189].Di;
	bConnectYourBitHere		:= IN_CU.tCustDigIn[190].Di;
	bConnectYourBitHere		:= IN_CU.tCustDigIn[191].Di;
	bConnectYourBitHere		:= IN_CU.tCustDigIn[192].Di;

	(* reserve digital input 193 *)
	bConnectYourBitHere		:= IN_CU.tCustDigIn[193].Di;
	bConnectYourBitHere		:= IN_CU.tCustDigIn[194].Di;
	bConnectYourBitHere		:= IN_CU.tCustDigIn[195].Di;
	bConnectYourBitHere		:= IN_CU.tCustDigIn[196].Di;

	(* reserve digital input 197 *)
	bConnectYourBitHere		:= IN_CU.tCustDigIn[197].Di;
	bConnectYourBitHere		:= IN_CU.tCustDigIn[198].Di;
	bConnectYourBitHere		:= IN_CU.tCustDigIn[199].Di;

	(* reserve digital input 200 *)
	bConnectYourBitHere		:= IN_CU.tCustDigIn[200].Di;
	OUT_CU.bCustDigIn[200]	:= IN_CU.tCustDigIn[200].Di;												(*stated here as array size check only*)
	MM2VIS.bCustDigIn[200]	:= IN_CU.tCustDigIn[200].Di;												(*stated here as array size check only*)

	(*********************************************************************************************************************************)

//VORSCHLAG NEU:
	(********************************************************)
	(*                                                      *)
	(*                DIGITAL OUTPUT SECTION                *)
	(*                                                      *)
	(********************************************************)												bConnectYourBitHere		:= NOT bDigOut_Release_Default; 	(*please keep this line unchanged for debugging purpose. This keeps DO´s shut off per default*)

//	(* Reservedigitalausgang x *)								(* (KONFIGURATIONSBEISPIEL) *)
//	(* reserve digital output X *)								(* (CONFIGURATION EXAMPLE)  *)
//	(***************************)
//	OUT_CU.tCustDigOut[x].Do :=								   NOT IN_CU.bMsg[1056] AND  bConnectYourBitHere ;	(*Anpassen entsprechend Kundenanforderung*)			(* change customized *)
//																 		|					+-------------------(*hier eigene Variable einsetzen*)					(* change 'bConnectYourBitHere' customized *)
//																		+---------------------------------------(*hier NOT AUS bzw. Abstellung nicht vergessen*)	(* change E-Stop or alarm stop condition customized *)
//
//																							+-------------------(*Möglichkeit zur Anbindung Handbedienbene mit IN_CU.tManAuxCtr.bAuxCust[x] *)	(* change customized *)
//	MM2VIS.bCustDigOut[x]	:= OUT_CU.tCustDigOut[x].Do;														(*Dies Variabele iat für VIS Verwendung vorber.*)	(* change 'bConnectYourBitHere' customized *)

	(* reserve digital output 1 *)
	OUT_CU.tCustDigOut[1].Do :=		NOT IN_CU.bMsg[1056] AND  bConnectYourBitHere ;
	(* reserve digital output 2 *)
	OUT_CU.tCustDigOut[2].Do :=		NOT IN_CU.bMsg[1056] AND  bConnectYourBitHere ;
	(* reserve digital output 3 *)
//	OUT_CU.tCustDigOut[3].Do :=		NOT IN_CU.bMsg[1056] AND  bConnectYourBitHere ; 	(*VSofti*)
	(* reserve digital output 4 *)
	OUT_CU.tCustDigOut[4].Do :=		NOT IN_CU.bMsg[1056] AND  bConnectYourBitHere ;

	(* reserve digital output 5 *)
	OUT_CU.tCustDigOut[5].Do :=		NOT IN_CU.bMsg[1056] AND  bConnectYourBitHere ;
	(* reserve digital output 6 *)
//	OUT_CU.tCustDigOut[6].Do :=		NOT IN_CU.bMsg[1056] AND  bConnectYourBitHere ; 	(*VSofti*)
	(* reserve digital output 7 *)
	OUT_CU.tCustDigOut[7].Do :=		NOT IN_CU.bMsg[1056] AND  bConnectYourBitHere ;
	(* reserve digital output 8 *)
	OUT_CU.tCustDigOut[8].Do :=		NOT IN_CU.bMsg[1056] AND  bConnectYourBitHere ;

	(* reserve digital output 9 *)
	OUT_CU.tCustDigOut[9].Do :=		NOT IN_CU.bMsg[1056] AND  bConnectYourBitHere ;
	OUT_CU.tCustDigOut[10].Do :=	NOT IN_CU.bMsg[1056] AND  bConnectYourBitHere ;
	OUT_CU.tCustDigOut[11].Do :=	NOT IN_CU.bMsg[1056] AND  bConnectYourBitHere ;
	OUT_CU.tCustDigOut[12].Do :=	NOT IN_CU.bMsg[1056] AND  bConnectYourBitHere ;

	(* reserve digital output 13 *)
	OUT_CU.tCustDigOut[13].Do :=	NOT IN_CU.bMsg[1056] AND  bConnectYourBitHere ;
	OUT_CU.tCustDigOut[14].Do :=	NOT IN_CU.bMsg[1056] AND  bConnectYourBitHere ;
	OUT_CU.tCustDigOut[15].Do :=	NOT IN_CU.bMsg[1056] AND  bConnectYourBitHere ;
//	OUT_CU.tCustDigOut[16].Do :=	NOT IN_CU.bMsg[1056] AND  bConnectYourBitHere ; 	(*VSofti*)

	(* reserve digital output 17 *)
//	OUT_CU.tCustDigOut[17].Do :=	NOT IN_CU.bMsg[1056] AND  bConnectYourBitHere ; 	(*VSofti*)
//	OUT_CU.tCustDigOut[18].Do :=	NOT IN_CU.bMsg[1056] AND  bConnectYourBitHere ; 	(*VSofti*)
//	OUT_CU.tCustDigOut[19].Do :=	NOT IN_CU.bMsg[1056] AND  bConnectYourBitHere ; 	(*VSofti*)
//	OUT_CU.tCustDigOut[20].Do :=	NOT IN_CU.bMsg[1056] AND  bConnectYourBitHere ; 	(*VSofti*)

	(* reserve digital output 21 *)
//	OUT_CU.tCustDigOut[21].Do :=	NOT IN_CU.bMsg[1056] AND  bConnectYourBitHere ; 	(*VSofti*)
//	OUT_CU.tCustDigOut[22].Do :=	NOT IN_CU.bMsg[1056] AND  bConnectYourBitHere ; 	(*VSofti*)
//	OUT_CU.tCustDigOut[23].Do :=	NOT IN_CU.bMsg[1056] AND  bConnectYourBitHere ; 	(*VSofti*)
	OUT_CU.tCustDigOut[24].Do :=	NOT IN_CU.bMsg[1056] AND  bConnectYourBitHere ;

	(* reserve digital output 25 *)
	OUT_CU.tCustDigOut[25].Do :=	NOT IN_CU.bMsg[1056] AND  bConnectYourBitHere ;
//	OUT_CU.tCustDigOut[26].Do :=	NOT IN_CU.bMsg[1056] AND  bConnectYourBitHere ; 	(*VSofti*)
//	OUT_CU.tCustDigOut[27].Do :=	NOT IN_CU.bMsg[1056] AND  bConnectYourBitHere ; 	(*VSofti*)
//	OUT_CU.tCustDigOut[28].Do :=	NOT IN_CU.bMsg[1056] AND  bConnectYourBitHere ; 	(*VSofti*)

	(* reserve digital output 31 *)
//	OUT_CU.tCustDigOut[29].Do :=	NOT IN_CU.bMsg[1056] AND  bConnectYourBitHere ; 	(*VSofti*)
//	OUT_CU.tCustDigOut[30].Do :=	NOT IN_CU.bMsg[1056] AND  bConnectYourBitHere ; 	(*VSofti*)
	OUT_CU.tCustDigOut[31].Do :=	NOT IN_CU.bMsg[1056] AND  bConnectYourBitHere ;
	OUT_CU.tCustDigOut[32].Do :=	NOT IN_CU.bMsg[1056] AND  bConnectYourBitHere ;

	(* reserve digital output 33 *)
	OUT_CU.tCustDigOut[33].Do :=	NOT IN_CU.bMsg[1056] AND  bConnectYourBitHere ;
	OUT_CU.tCustDigOut[34].Do :=	NOT IN_CU.bMsg[1056] AND  bConnectYourBitHere ;
//	OUT_CU.tCustDigOut[35].Do :=	NOT IN_CU.bMsg[1056] AND  bConnectYourBitHere ; 	(*VSofti*)
//	OUT_CU.tCustDigOut[36].Do :=	NOT IN_CU.bMsg[1056] AND  bConnectYourBitHere ; 	(*VSofti*)

	(* reserve digital output 37 *)
//	OUT_CU.tCustDigOut[37].Do :=	NOT IN_CU.bMsg[1056] AND  bConnectYourBitHere ; 	(*VSofti*)
//	OUT_CU.tCustDigOut[38].Do :=	NOT IN_CU.bMsg[1056] AND  bConnectYourBitHere ; 	(*VSofti*)
//	OUT_CU.tCustDigOut[39].Do :=	NOT IN_CU.bMsg[1056] AND  bConnectYourBitHere ; 	(*VSofti*)
//	OUT_CU.tCustDigOut[40].Do :=	NOT IN_CU.bMsg[1056] AND  bConnectYourBitHere ; 	(*VSofti*)

	(* reserve digital output 41 *)
//	OUT_CU.tCustDigOut[41].Do :=	NOT IN_CU.bMsg[1056] AND  bConnectYourBitHere ; 	(*VSofti*)
//	OUT_CU.tCustDigOut[42].Do :=	NOT IN_CU.bMsg[1056] AND  bConnectYourBitHere ; 	(*VSofti*)
//	OUT_CU.tCustDigOut[43].Do :=	NOT IN_CU.bMsg[1056] AND  bConnectYourBitHere ; 	(*VSofti*)
//	OUT_CU.tCustDigOut[44].Do :=	NOT IN_CU.bMsg[1056] AND  bConnectYourBitHere ; 	(*VSofti*)

	(* reserve digital output 45 *)
//	OUT_CU.tCustDigOut[45].Do :=	NOT IN_CU.bMsg[1056] AND  bConnectYourBitHere ; 	(*VSofti*)
//	OUT_CU.tCustDigOut[46].Do :=	NOT IN_CU.bMsg[1056] AND  bConnectYourBitHere ; 	(*VSofti*)
	OUT_CU.tCustDigOut[47].Do :=	NOT IN_CU.bMsg[1056] AND  bConnectYourBitHere ;
//	OUT_CU.tCustDigOut[48].Do :=	NOT IN_CU.bMsg[1056] AND  bConnectYourBitHere ; 	(*VSofti*)

	(* reserve digital output 49 *)
//	OUT_CU.tCustDigOut[49].Do :=	NOT IN_CU.bMsg[1056] AND  bConnectYourBitHere ; 	(*VSofti*)
//	OUT_CU.tCustDigOut[50].Do :=	NOT IN_CU.bMsg[1056] AND  bConnectYourBitHere ; 	(*VSofti*)
	OUT_CU.tCustDigOut[51].Do :=	NOT IN_CU.bMsg[1056] AND  bConnectYourBitHere ;
	OUT_CU.tCustDigOut[52].Do :=	NOT IN_CU.bMsg[1056] AND  bConnectYourBitHere ;

	(* reserve digital output 53 *)
	OUT_CU.tCustDigOut[53].Do :=	NOT IN_CU.bMsg[1056] AND  bConnectYourBitHere ;
	OUT_CU.tCustDigOut[54].Do :=	NOT IN_CU.bMsg[1056] AND  bConnectYourBitHere ;
	OUT_CU.tCustDigOut[55].Do :=	NOT IN_CU.bMsg[1056] AND  bConnectYourBitHere ;
	OUT_CU.tCustDigOut[56].Do :=	NOT IN_CU.bMsg[1056] AND  bConnectYourBitHere ;

	(* reserve digital output 57 *)
	OUT_CU.tCustDigOut[57].Do :=	NOT IN_CU.bMsg[1056] AND  bConnectYourBitHere ;
	OUT_CU.tCustDigOut[58].Do :=	NOT IN_CU.bMsg[1056] AND  bConnectYourBitHere ;
	OUT_CU.tCustDigOut[59].Do :=	NOT IN_CU.bMsg[1056] AND  bConnectYourBitHere ;
	OUT_CU.tCustDigOut[60].Do :=	NOT IN_CU.bMsg[1056] AND  bConnectYourBitHere ;

	(* reserve digital output 61 *)
	OUT_CU.tCustDigOut[61].Do :=	NOT IN_CU.bMsg[1056] AND  bConnectYourBitHere ;
	OUT_CU.tCustDigOut[62].Do :=	NOT IN_CU.bMsg[1056] AND  bConnectYourBitHere ;
	OUT_CU.tCustDigOut[63].Do :=	NOT IN_CU.bMsg[1056] AND  bConnectYourBitHere ;
	OUT_CU.tCustDigOut[64].Do :=	NOT IN_CU.bMsg[1056] AND  bConnectYourBitHere ;

	(* reserve digital output 65 *)
	OUT_CU.tCustDigOut[65].Do :=	NOT IN_CU.bMsg[1056] AND  bConnectYourBitHere ;
	OUT_CU.tCustDigOut[66].Do :=	NOT IN_CU.bMsg[1056] AND  bConnectYourBitHere ;
	OUT_CU.tCustDigOut[67].Do :=	NOT IN_CU.bMsg[1056] AND  bConnectYourBitHere ;
	OUT_CU.tCustDigOut[68].Do :=	NOT IN_CU.bMsg[1056] AND  bConnectYourBitHere ;

	(* reserve digital output 69 *)
	OUT_CU.tCustDigOut[69].Do :=	NOT IN_CU.bMsg[1056] AND  bConnectYourBitHere ;
	OUT_CU.tCustDigOut[70].Do :=	NOT IN_CU.bMsg[1056] AND  bConnectYourBitHere ;
	OUT_CU.tCustDigOut[71].Do :=	NOT IN_CU.bMsg[1056] AND  bConnectYourBitHere ;
	OUT_CU.tCustDigOut[72].Do :=	NOT IN_CU.bMsg[1056] AND  bConnectYourBitHere ;

	(* reserve digital output 73 *)
	OUT_CU.tCustDigOut[73].Do :=	NOT IN_CU.bMsg[1056] AND  bConnectYourBitHere ;
	OUT_CU.tCustDigOut[74].Do :=	NOT IN_CU.bMsg[1056] AND  bConnectYourBitHere ;
	OUT_CU.tCustDigOut[75].Do :=	NOT IN_CU.bMsg[1056] AND  bConnectYourBitHere ;
	OUT_CU.tCustDigOut[76].Do :=	NOT IN_CU.bMsg[1056] AND  bConnectYourBitHere ;

	(* reserve digital output 77 *)
	OUT_CU.tCustDigOut[77].Do :=	NOT IN_CU.bMsg[1056] AND  bConnectYourBitHere ;
	OUT_CU.tCustDigOut[78].Do :=	NOT IN_CU.bMsg[1056] AND  bConnectYourBitHere ;
	OUT_CU.tCustDigOut[79].Do :=	NOT IN_CU.bMsg[1056] AND  bConnectYourBitHere ;
	OUT_CU.tCustDigOut[80].Do :=	NOT IN_CU.bMsg[1056] AND  bConnectYourBitHere ;

	(* reserve digital output 81 *)
	OUT_CU.tCustDigOut[81].Do :=	NOT IN_CU.bMsg[1056] AND  bConnectYourBitHere ;
	OUT_CU.tCustDigOut[82].Do :=	NOT IN_CU.bMsg[1056] AND  bConnectYourBitHere ;
	OUT_CU.tCustDigOut[83].Do :=	NOT IN_CU.bMsg[1056] AND  bConnectYourBitHere ;
	OUT_CU.tCustDigOut[84].Do :=	NOT IN_CU.bMsg[1056] AND  bConnectYourBitHere ;

	(* reserve digital output 85 *)
	OUT_CU.tCustDigOut[85].Do :=	NOT IN_CU.bMsg[1056] AND  bConnectYourBitHere ;
	OUT_CU.tCustDigOut[86].Do :=	NOT IN_CU.bMsg[1056] AND  bConnectYourBitHere ;
	OUT_CU.tCustDigOut[87].Do :=	NOT IN_CU.bMsg[1056] AND  bConnectYourBitHere ;
	OUT_CU.tCustDigOut[88].Do :=	NOT IN_CU.bMsg[1056] AND  bConnectYourBitHere ;

	(* reserve digital output 89 *)
	OUT_CU.tCustDigOut[89].Do :=	NOT IN_CU.bMsg[1056] AND  bConnectYourBitHere ;
	OUT_CU.tCustDigOut[90].Do :=	NOT IN_CU.bMsg[1056] AND  bConnectYourBitHere ;
	OUT_CU.tCustDigOut[91].Do :=	NOT IN_CU.bMsg[1056] AND  bConnectYourBitHere ;
	OUT_CU.tCustDigOut[92].Do :=	NOT IN_CU.bMsg[1056] AND  bConnectYourBitHere ;

	(* reserve digital output 93 *)
	OUT_CU.tCustDigOut[93].Do :=	NOT IN_CU.bMsg[1056] AND  bConnectYourBitHere ;
	OUT_CU.tCustDigOut[94].Do :=	NOT IN_CU.bMsg[1056] AND  bConnectYourBitHere ;
	OUT_CU.tCustDigOut[95].Do :=	NOT IN_CU.bMsg[1056] AND  bConnectYourBitHere ;
	OUT_CU.tCustDigOut[96].Do :=	NOT IN_CU.bMsg[1056] AND  bConnectYourBitHere ;

	(* reserve digital output 97 *)
	OUT_CU.tCustDigOut[97].Do :=	NOT IN_CU.bMsg[1056] AND  bConnectYourBitHere ;
	OUT_CU.tCustDigOut[98].Do :=	NOT IN_CU.bMsg[1056] AND  bConnectYourBitHere ;
	OUT_CU.tCustDigOut[99].Do :=	NOT IN_CU.bMsg[1056] AND  bConnectYourBitHere ;
	OUT_CU.tCustDigOut[100].Do :=	NOT IN_CU.bMsg[1056] AND  bConnectYourBitHere ;

	(* reserve digital output 101 *)
	OUT_CU.tCustDigOut[101].Do :=	NOT IN_CU.bMsg[1056] AND  bConnectYourBitHere ;
	OUT_CU.tCustDigOut[102].Do :=	NOT IN_CU.bMsg[1056] AND  bConnectYourBitHere ;
	OUT_CU.tCustDigOut[103].Do :=	NOT IN_CU.bMsg[1056] AND  bConnectYourBitHere ;
	OUT_CU.tCustDigOut[104].Do :=	NOT IN_CU.bMsg[1056] AND  bConnectYourBitHere ;

	(* reserve digital output 105 *)
	OUT_CU.tCustDigOut[105].Do :=	NOT IN_CU.bMsg[1056] AND  bConnectYourBitHere ;
	OUT_CU.tCustDigOut[106].Do :=	NOT IN_CU.bMsg[1056] AND  bConnectYourBitHere ;
	OUT_CU.tCustDigOut[107].Do :=	NOT IN_CU.bMsg[1056] AND  bConnectYourBitHere ;
	OUT_CU.tCustDigOut[108].Do :=	NOT IN_CU.bMsg[1056] AND  bConnectYourBitHere ;

	(* reserve digital output 109 *)
	OUT_CU.tCustDigOut[109].Do :=	NOT IN_CU.bMsg[1056] AND  bConnectYourBitHere ;
	OUT_CU.tCustDigOut[110].Do :=	NOT IN_CU.bMsg[1056] AND  bConnectYourBitHere ;
	OUT_CU.tCustDigOut[111].Do :=	NOT IN_CU.bMsg[1056] AND  bConnectYourBitHere ;
	OUT_CU.tCustDigOut[112].Do :=	NOT IN_CU.bMsg[1056] AND  bConnectYourBitHere ;

	(* reserve digital output 113 *)
	OUT_CU.tCustDigOut[113].Do :=	NOT IN_CU.bMsg[1056] AND  bConnectYourBitHere ;
	OUT_CU.tCustDigOut[114].Do :=	NOT IN_CU.bMsg[1056] AND  bConnectYourBitHere ;
	OUT_CU.tCustDigOut[115].Do :=	NOT IN_CU.bMsg[1056] AND  bConnectYourBitHere ;
	OUT_CU.tCustDigOut[116].Do :=	NOT IN_CU.bMsg[1056] AND  bConnectYourBitHere ;

	(* reserve digital output 117 *)
	OUT_CU.tCustDigOut[117].Do :=	NOT IN_CU.bMsg[1056] AND  bConnectYourBitHere ;
	OUT_CU.tCustDigOut[118].Do :=	NOT IN_CU.bMsg[1056] AND  bConnectYourBitHere ;
	OUT_CU.tCustDigOut[119].Do :=	NOT IN_CU.bMsg[1056] AND  bConnectYourBitHere ;
	OUT_CU.tCustDigOut[120].Do :=	NOT IN_CU.bMsg[1056] AND  bConnectYourBitHere ;

	(**********************************************)
	(*****      END OF CONFIGURATION AREA     *****)
	(**********************************************)

	(*+++++ NO CHANGES BEJOND THIS LINE! +++++++++*)

	(* prepard copy process *)
	FOR cnt := 1 TO 200 DO
		(*forward value to module output for use in other modules*)
		OUT_CU.bCustDigIn[cnt]	:= IN_CU.tCustDigIn[cnt].Di;	(* prepared for possible usage in other modules *)
	END_FOR
	(* prepard copy process *)
	FOR cnt := 1 TO 150 DO
		(*forward value to module output for use in other modules*)
		OUT_CU.bCustDigOut[cnt] := OUT_CU.tCustDigOut[cnt].Do;	(* Copy to DO structure; bCustDigOut is also prepared for possible usage in other modules *)
	END_FOR

	(*forward value to visualisation output*)
	MM2VIS.bCustDigIn :=		OUT_CU.bCustDigIn		;
	MM2VIS.bCustDigOut :=		OUT_CU.bCustDigOut		;	(*Fehlt noch*)

	(*Bugfix Version for missing VIS parameter: Set all DigOut as active*)
	//	TON_DigOut.IN := ( IN_CU.tPB2MM.bSys_Run  AND bDigOut_Release_Default );
//	TON_DigOut(PT := T#10s);
//	R_TRIG_DigOut(CLK:=TON_DigOut.Q);
	IF bDigOut_Release_Default THEN	 //IF	bBugfix_CustDigOut_Active THEN
		FOR cnt := 1 TO 150 DO
		(*Bugfix *)   Para.bCustDigOut_Active[cnt]		:= bDigOut_Release_Default; 	(*set parameter value directly*)
		END_FOR
	END_IF

END_PROGRAM
```

#### c_digInit.st
```iecst
(*******************************************************************************
CUSTOMIZED: c_dig.st - connection and processing of prepared digital I /O channels (cyclic)

This code is confidential and proprietary to the INNIO Company.
It may not be used in any form, or reproduced in any manner, without the express
written permission of the INNIO Company.
Copyright, INNIO Company, 2019

Customized modifications: -
------------------------

History:
-------
V0.1	05-03-2002	Weitzer, generated from zaehler.c / V0.1
...
V4.02.0 24.06.2015	Zengerer cleanup

Instructions for use:
--------------------

Outstandings:
------------

*******************************************************************************)

PROGRAM _INIT

	(* ...	change or extend this init file customized, if needed.	*)																						bConnectYourBitHere;		(* this statements mark places all over the code, where you shoud replace it with your own variable names according to customer needs; but please leaf this single occurence unchanged for internal purposes*)

	bDigOut_Release_Default := TRUE; 	(*bDigOut_Release_Default = 1 == alle DO Kanäle sind vordefiniert als aktiv, 0= alle DO Parameter werden DISABELED als default*)

	(**********************************************)
	(*****      END OF CONFIGURATION AREA     *****)
	(**********************************************)
	(* NO CHANGES BEJOND THIS LINE! *)

	(*BETAversion, Abklärung fehlt noch*)	(*bDigOut_Release_Default = 1 == alle DO Kanäle sind vordefiniert als aktiv, 0= alle DO Parameter werden DISABELED als default*)
	FOR cnt := 1 TO 150 DO
		ParaFactoryDefault.bCustDigOut_Active[cnt]		:= bDigOut_Release_Default; 	(*set default parameter value only*)
	END_FOR

END_PROGRAM
```

#### c_dig.var
```iecst
VAR
	bConnectYourBitHere : BOOL := FALSE; (*Dummy Bit to be replaced by plant specific variable*)
	bDigOut_Release_Default : BOOL; (*1=Alle DO sind vordefiniert aktiv, 0= alle DO Parameter werden DISABELED als default*)
END_VAR
```

### Program Logical/Customized/c_aux (IEC, version 4.13.0) - customisation task for auxiliaries display page on VIS

#### c_auxCyclic.st
```iecst
(*******************************************************************************
c_aux 			customized auxiliaries #21-30 for visualization

This code is confidential and proprietary to the INNIO Company.
It may not be used in any form, or reproduced in any manner,
without written permission of the INNIO Company.
Copyright, INNIO Company, 2022

Customized modifications: -
------------------------

History:
-------
V3.20.0	14-10-2010 lettenb.	new, function moved from fb31_hb
V3.21	04.09.2013 zengerer _Active typ changed to INT (entspr. DianeWIN Version)
V3.22	12.09.2013 zengerer MM2Vis added
V4.00.1	09.05.2014 zengerer	do no predefinition for parameter values, this causes VIS troubles!
				 			beta bugfix: reduced Para update speed to hardcoded defaults with 'bSetFixParaToDefault' bit to avoid VIS troubles with hardcoded para values
							bEC_Rel, bChC_Rel included from MM_HC
V4.04.0	08.11.2016 lettenb.	OUT_CU.bEC_Rel: Para.bAuxEC_Visible added(stary)
V4.07.0	09.08.2018 Schmid	2nd low temperature charge cooling circuit added (bChC2_Rel)
V4.07.0	27.02.2019 zengerer remove parameter preparation, beta defaults with 'bSetFixParaToDefault' removed
V4.11.0	17.12.2021 Schmid	control battery check
		20.01.2022 zengerer Reintegrate Customer Extention Package
V4.11.1	14.02.2022 Schmid	GoodQual default TRUE for control battery check supply monitoring
		23.02.2022 lettenb. OUT_CU.bChC_Rel: bMsg2117(charge cooler water pressure low) removed, request system owner, bugfix
V4.11.2	23.02.2022 Schmid	+M control battery check option removed - covered by buffer battery check (coordinated execution with starter battery check required)
V4.13.0	24.08.2023 Zengerer IN_CU.bMsg[xxxx] introduced

Instructions for use:
--------------------
connect var for display customized auxiliaries
AVOID HARDCODED PARAMETER VALUES! Set display typ of each aux in parameter file.

Outstandings:
------------
bSetFixParaToDefault?

*******************************************************************************)
PROGRAM _CYCLIC
	(*------------------------------------------------------------------------------------------*)
	(* release emergency cooler from monitoring (remove not applicable parts) (ex K_frg) *)
	OUT_CU.bEC_Rel 	:=  NOT IN_CU.bMsg[1031]
			        AND NOT IN_CU.bMsg[1053]
					AND NOT IN_CU.bMsg[1054]
					AND NOT IN_CU.bMsg[3404]
					AND(NOT IN_CU.bMsg[2117] OR Para.bAuxEC_Visible) (* for EngineVis >= 2.5.x *)
					AND NOT IN_CU.bMsg[1019];

	(* release charge cooler from monitoring (remove not applicable parts) (ex GK_frg) *)
	OUT_CU.bChC_Rel	:=  NOT IN_CU.bMsg[1031]
					AND NOT IN_CU.bMsg[1053]
					AND NOT IN_CU.bMsg[1054];

	(* release charge cooler 2 from monitoring (remove not applicable parts) *)
	OUT_CU.bChC2_Rel	:=  NOT IN_CU.bMsg[1031]
						AND NOT IN_CU.bMsg[1053]
						AND NOT IN_CU.bMsg[1054]
						AND NOT IN_CU.bMsg[9226];

	(*------------------------------------------------------------------------------------------*)
	(* control battery voltage check *)
	iOptLocation_CtrlBatMon[1]	:=	1;		// set index variable according to position of battery test set
	iOptLocation_CtrlBatMon[2]	:=	2;		// predefined options: 1: +A / 2: +AUX1 / 3: +AUX2 / 4: +CUSTOM
	iOptLocation_CtrlBatMon[3]	:=	3;		// not used test sets can remain in default setting - GoodQual detects usage automatically
	iOptLocation_CtrlBatMon[4]	:=	4;		// for customization see instructions below

	(*iOptLocation_CtrlBatMon contains the location of control battery test sets (control cabinets)
	In the preconfigured status, in position 1 there is the measure +A, in position 2 the measure +AUX1, in position 2 the measure +AUX2 and in position 4 the measure +CUSTOM
	For example, when iOptLocation_CtrlBatMon = [2,1,3,4], in position 1 there is the measure +AUX1, in position 2 the measure +A, in position 3 the measure +AUX2 and in position 4 the measure +CUSTOM
	*)

	FOR iIdx_CtrlBatMon := 1 TO iNum_CtrlBatMon DO
		CASE iOptLocation_CtrlBatMon[iIdx_CtrlBatMon] OF
			1:	(* +A *)
				OUT_CU.sLocIdent_CtrlBatMon[iIdx_CtrlBatMon]	:=	'+A';																// control cabinet location of test set
				OUT_CU.bAuxV_ok_CtrlBatMon[iIdx_CtrlBatMon]		:=	IN_CU.tAuxV_Supply_Ok.Di	OR NOT IN_CU.tAuxV_Supply_Ok.GoodQual;	// according supply voltage status

			2:	(* +AUX1 *)
				OUT_CU.sLocIdent_CtrlBatMon[iIdx_CtrlBatMon]	:=	'+AUX1';
				OUT_CU.bAuxV_ok_CtrlBatMon[iIdx_CtrlBatMon]		:=	IN_CU.tAuxV_Aux_ok.Di		OR NOT IN_CU.tAuxV_Aux_ok.GoodQual;

			3:	(* +AUX2 *)
				OUT_CU.sLocIdent_CtrlBatMon[iIdx_CtrlBatMon]	:=	'+AUX2';
				OUT_CU.bAuxV_ok_CtrlBatMon[iIdx_CtrlBatMon]		:=	IN_CU.tAuxV_Aux_ok.Di		OR NOT IN_CU.tAuxV_Aux_ok.GoodQual;

			4:	(* +CUSTOM *)
				OUT_CU.sLocIdent_CtrlBatMon[iIdx_CtrlBatMon]	:=	'+CUSTOM';
				OUT_CU.bAuxV_ok_CtrlBatMon[iIdx_CtrlBatMon]		:=	FALSE;	//IN_CU.tAuxV_CUSTOM_ok.Di OR NOT IN_CU.tAuxV_CUSTOM_ok.GoodQual;
		END_CASE;
	END_FOR;

	(* if customized adjustments (location, voltage supply) are required, overwrite elements in the following: *)
	//	OUT_CU.sLocIdent_CtrlBatMon[1..4]	:=	'+XYZ';
	//	OUT_CU.bAuxV_ok_CtrlBatMon[1..4]	:=	IN_CU.tAuxV_CUSTOM_ok.Di OR NOT IN_CU.tAuxV_CUSTOM_ok.GoodQual;

	(*------------------------------------------------------------------------------------------*)

	OUT_CU.bAuxCust_Dem[1]	;//:=	FALSE;		(* reserve auxiliary  #1 		*)		(* Connect your customisation variable here; VIS: customize texts! *)
	(*Hint: Set VIS appearance with Para.iAuxCust_Active[1]:	 0=invisible, 1=ON/OFF, 2=OPEN/CLOSED	*)	(* 0=keine Anzeige, 1=EIN/AUS, 2=OFFEN/GESCHLOSSEN) *)
	(*IN_CU.tManAuxCtr.bAuxCust[x] 1-10 prepared *)	(* change customized *)

	OUT_CU.bAuxCust_Dem[2]	;//:=	FALSE;		(* reserve auxiliary  #2 		*)		(* Connect your customisation variable here; VIS: customize texts! *)

	OUT_CU.bAuxCust_Dem[3]	;//:=	FALSE;		(* reserve auxiliary  #3 		*)		(* Connect your customisation variable here; VIS: customize texts! *)

	OUT_CU.bAuxCust_Dem[4]	;//:=	FALSE;		(* reserve auxiliary  #4 		*)

	OUT_CU.bAuxCust_Dem[5]	;//:=	FALSE;		(* reserve auxiliary  #5 		*)

	OUT_CU.bAuxCust_Dem[6]	;//:=	FALSE;		(* reserve auxiliary  #6 		*)

	OUT_CU.bAuxCust_Dem[7]	;//:=	FALSE;		(* reserve auxiliary  #7 		*)

	OUT_CU.bAuxCust_Dem[8]	;//:=	FALSE;		(* reserve auxiliary  #8 		*)

	OUT_CU.bAuxCust_Dem[9]	;//:=	FALSE;		(* reserve auxiliary  #9 		*)

	OUT_CU.bAuxCust_Dem[10]	;//:=	FALSE;		(* reserve auxiliary  #10		*)

	OUT_CU.bAuxCust_Dem[11]	;//:=	FALSE;		(* reserve auxiliary #11 		*)

	OUT_CU.bAuxCust_Dem[12]	;//:=	FALSE;		(* reserve auxiliary #12 		*)

	OUT_CU.bAuxCust_Dem[13]	;//:=	FALSE;		(* reserve auxiliary #13 		*)

	OUT_CU.bAuxCust_Dem[14]	;//:=	FALSE;		(* reserve auxiliary #14 		*)

	OUT_CU.bAuxCust_Dem[15]	;//:=	FALSE;		(* reserve auxiliary #15 		*)

	OUT_CU.bAuxCust_Dem[16]	;//:=	FALSE;		(* reserve auxiliary #16 		*)

	OUT_CU.bAuxCust_Dem[17]	;//:=	FALSE;		(* reserve auxiliary #17 		*)

	OUT_CU.bAuxCust_Dem[18]	;//:=	FALSE;		(* reserve auxiliary #18 		*)

	OUT_CU.bAuxCust_Dem[19]	;//:=	FALSE;		(* reserve auxiliary #19 		*)

	OUT_CU.bAuxCust_Dem[20]	;//:=	FALSE;		(* reserve auxiliary #20 		*)

	OUT_CU.bAuxCust_Dem[21]	;//:=	FALSE;		(* reserve auxiliary #21 		*)
	(*Hint: Set VIS aperance with Para.iAuxCust_Active[21]:	 0=invisible, 1=ON/OFF, 2=OPEN/CLOSED	*)	(* 0=keine Anzeige, 1=EIN/AUS, 2=OFFEN/GESCHLOSSEN) *)

	OUT_CU.bAuxCust_Dem[22]	;//:=	FALSE;		(* reserve auxiliary #22 		*)

	OUT_CU.bAuxCust_Dem[23]	;//:=	FALSE;		(* reserve auxiliary #23 		*)

	OUT_CU.bAuxCust_Dem[24]	;//:=	FALSE;		(* reserve auxiliary #24		*)

	OUT_CU.bAuxCust_Dem[25]	;//:=	FALSE;		(* reserve auxiliary #25 		*)

	OUT_CU.bAuxCust_Dem[26]	;//:=	FALSE;		(* reserve auxiliary #26 		*)

	OUT_CU.bAuxCust_Dem[27]	;//:=	FALSE;		(* reserve auxiliary #27 		*)

	OUT_CU.bAuxCust_Dem[28]	;//:=	FALSE;		(* reserve auxiliary #28 		*)

	OUT_CU.bAuxCust_Dem[29]	;//:=	FALSE;		(* reserve auxiliary #29 		*)

	OUT_CU.bAuxCust_Dem[30]	;//:=	FALSE;		(* reserve auxiliary #30 		*)

	OUT_CU.bAuxCust_Dem[31]	;//:=	FALSE;		(* reserve auxiliary #31 		*)

	OUT_CU.bAuxCust_Dem[32]	;//:=	FALSE;		(* reserve auxiliary #32 		*)

	OUT_CU.bAuxCust_Dem[33]	;//:=	FALSE;		(* reserve auxiliary #33 		*)

	OUT_CU.bAuxCust_Dem[34]	;//:=	FALSE;		(* reserve auxiliary #34		*)

	OUT_CU.bAuxCust_Dem[35]	;//:=	FALSE;		(* reserve auxiliary #35 		*)

	OUT_CU.bAuxCust_Dem[36]	;//:=	FALSE;		(* reserve auxiliary #36 		*)

	OUT_CU.bAuxCust_Dem[37]	;//:=	FALSE;		(* reserve auxiliary #37 		*)

	OUT_CU.bAuxCust_Dem[38]	;//:=	FALSE;		(* reserve auxiliary #38 		*)

	OUT_CU.bAuxCust_Dem[39]	;//:=	FALSE;		(* reserve auxiliary #39 		*)

	OUT_CU.bAuxCust_Dem[40]	;//:=	FALSE;		(* reserve auxiliary #40 		*)
	(*Hint: Set VIS aperance with Para.iAuxCust_Active[40]:	 0=invisible, 1=ON/OFF, 2=OPEN/CLOSED	*)	(* 0=keine Anzeige, 1=EIN/AUS, 2=OFFEN/GESCHLOSSEN) *)

	(*** DEFAULT CONFIG END ********************************************************************************************************)
	(*** DEFAULT CONFIG END  - ADD VIS EXTENTION PACKAGE also, to use more than the default number of channels *********************)
	(*** DEFAULT CONFIG END ********************************************************************************************************)

	OUT_CU.bAuxCust_Dem[41];//:=	FALSE;		(* reserve auxiliary #41		*) 	(*import HMI Extension *)
	OUT_CU.bAuxCust_Dem[42];//:=	FALSE;		(* reserve auxiliary #42		*) 	(*import HMI Extension *)
	OUT_CU.bAuxCust_Dem[43];//:=	FALSE;		(* reserve auxiliary #43		*) 	(*import HMI Extension *)
	OUT_CU.bAuxCust_Dem[44];//:=	FALSE;		(* reserve auxiliary #44		*) 	(*import HMI Extension *)
	OUT_CU.bAuxCust_Dem[45];//:=	FALSE;		(* reserve auxiliary #45		*) 	(*import HMI Extension *)
	OUT_CU.bAuxCust_Dem[46];//:=	FALSE;		(* reserve auxiliary #46		*) 	(*import HMI Extension *)
	OUT_CU.bAuxCust_Dem[47];//:=	FALSE;		(* reserve auxiliary #47		*) 	(*import HMI Extension *)
	OUT_CU.bAuxCust_Dem[48];//:=	FALSE;		(* reserve auxiliary #48		*) 	(*import HMI Extension *)
	OUT_CU.bAuxCust_Dem[49];//:=	FALSE;		(* reserve auxiliary #49		*) 	(*import HMI Extension *)

	OUT_CU.bAuxCust_Dem[50];//:=	FALSE;		(* reserve auxiliary #50		*) 	(*import HMI Extension *)
	OUT_CU.bAuxCust_Dem[51];//:=	FALSE;		(* reserve auxiliary #51		*) 	(*import HMI Extension *)
	OUT_CU.bAuxCust_Dem[52];//:=	FALSE;		(* reserve auxiliary #52		*) 	(*import HMI Extension *)
	OUT_CU.bAuxCust_Dem[53];//:=	FALSE;		(* reserve auxiliary #53		*) 	(*import HMI Extension *)
	OUT_CU.bAuxCust_Dem[54];//:=	FALSE;		(* reserve auxiliary #54		*) 	(*import HMI Extension *)
	OUT_CU.bAuxCust_Dem[55];//:=	FALSE;		(* reserve auxiliary #55		*) 	(*import HMI Extension *)
	OUT_CU.bAuxCust_Dem[56];//:=	FALSE;		(* reserve auxiliary #56		*) 	(*import HMI Extension *)
	OUT_CU.bAuxCust_Dem[57];//:=	FALSE;		(* reserve auxiliary #57		*) 	(*import HMI Extension *)
	OUT_CU.bAuxCust_Dem[58];//:=	FALSE;		(* reserve auxiliary #58		*) 	(*import HMI Extension *)
	OUT_CU.bAuxCust_Dem[59];//:=	FALSE;		(* reserve auxiliary #59		*) 	(*import HMI Extension *)

	OUT_CU.bAuxCust_Dem[60];//:=	FALSE;		(* reserve auxiliary #60		*) 	(*import HMI Extension *)
	OUT_CU.bAuxCust_Dem[61];//:=	FALSE;		(* reserve auxiliary #61		*) 	(*import HMI Extension *)
	OUT_CU.bAuxCust_Dem[62];//:=	FALSE;		(* reserve auxiliary #62		*) 	(*import HMI Extension *)
	OUT_CU.bAuxCust_Dem[63];//:=	FALSE;		(* reserve auxiliary #63		*) 	(*import HMI Extension *)
	OUT_CU.bAuxCust_Dem[64];//:=	FALSE;		(* reserve auxiliary #64		*) 	(*import HMI Extension *)
	OUT_CU.bAuxCust_Dem[65];//:=	FALSE;		(* reserve auxiliary #65		*) 	(*import HMI Extension *)
	OUT_CU.bAuxCust_Dem[66];//:=	FALSE;		(* reserve auxiliary #66		*) 	(*import HMI Extension *)
	OUT_CU.bAuxCust_Dem[67];//:=	FALSE;		(* reserve auxiliary #67		*) 	(*import HMI Extension *)
	OUT_CU.bAuxCust_Dem[68];//:=	FALSE;		(* reserve auxiliary #68		*) 	(*import HMI Extension *)
	OUT_CU.bAuxCust_Dem[69];//:=	FALSE;		(* reserve auxiliary #69		*) 	(*import HMI Extension *)

	OUT_CU.bAuxCust_Dem[70];//:=	FALSE;		(* reserve auxiliary #70		*) 	(*import HMI Extension *)

	(*------------------------------------------------------------------------------*)
	(*						  NO CHANGES BEJOND THIS LINE!			 				*)
	(*------------------------------------------------------------------------------*)

	MM2VIS.bAuxCust		 :=	OUT_CU.bAuxCust_Dem			;		(* forward status info to visualisation display (with check of exact matching array size) *)

	(*generate artificial parameter state changes - REMOVED *)

END_PROGRAM
```

#### c_aux.var
```iecst
VAR
	iOptLocation_CtrlBatMon : ARRAY[1..iNum_CtrlBatMon] OF USINT;
	iIdx_CtrlBatMon : USINT;
END_VAR
```

### Program Logical/Customized/c_coupl (IEC, version 4.14.0) - Bus Coupling IN/OUT data register
